(* CODESYS project CommonTypesAndFunctions.library
   Author: Stefan Dreyer
   Title: Common Helper for development
   Version: 1.0.0.0
   Placeholder: CommonTypsFunctions
   DocFormat: reStructuredText
   Description: Some things to collect...
      some based on OSCAT library.
      see www.oscat.de for here home
   Company: Stefan Dreyer
   LanguageModelAttribute: qualified-access-only
   DefaultNamespace: CommonTypesAndFunctions

Project tree, tasks and I/O mapping:
  libraries: CAA Types Extern, * (CAA Technical Workgroup); CAA Behaviour Model, * (CAA Technical Workgroup); CAA FB Factory, * (CAA Technical Workgroup); OSCAT NETWORK, 1.30 (OSCAT); SysSem, 3.5.5.0 (System); SysTypes Interfaces, 3.5.2.0 (System); BASIC, 3.3.3.0 (OSCAT); Time and Date, 3.5.7.0 (3S - Smart Software Solutions GmbH); CmpTls, 3.5.10.0 (System); SysProcess, 3.5.7.0 (System); SysTarget, 3.5.5.0 (System); SysMem, 3.5.12.0 (System); CmpX509Cert, 3.5.11.0 (System); CmpCrypto, 3.5.11.0 (System); MQTT, 1.1.0.0 (Stefan Dreyer); SysSocket2, 3.5.14.0 (System); SysSocket, 3.5.14.0 (System); Standard, 3.5.14.0 (System); CmpErrors2 Interfaces, 3.5.12.0 (System); Standard64, 3.5.13.0 (System)
  Common/
    Enums/
      data type ERROR
      data type VAR_TYPES
    Function Blocks/
      function block IP_CONTROL [ST]
      function block IP_CONTROL_135 [ST]
      function block IP_CONTROL_135_1 [ST]
      function block IP_CONTROL_old [ST]
      function block TIME_DATE_IMPULS [ST]
      function block TestString [ST]
      function block IP_CONTROL_TLS [ST]
      function block CounterToActuall [ST]: CounterInit, SetCounterResetImp
      function block StringImpact [ST]
      function block GetInstanceName [ST]: GetInstanceTopic
      function block RELAIS_OUT_16_TRANSLATOR [ST]
    Functions/
      function GET_DNS_IP [ST]
      function GetChar [ST]
      function find [ST]
      function len [ST]
      function concat [ST]
      function ResolveIPAddr [ST]
      function CheckDeltaValue [ST]
      function GetValueFromPointer [ST]
      function GetValueString [ST]
      function test [ST]
      function StrEquals [ST]
      function StrEqualsAtStart [ST]
      function GetValueFromStringPt [ST]
      function StrEqualsAtStartWithDelimiter [ST]
      function FindLastDot [ST]
      function MakeAllTypesPointer [ST]
      function GetJSONValue [ST]
    GlobalConstants/
      global variables MyConstants
    GlobalVariables/
      global variables Variables
    Interfaces/
    Structs/
    Templates/
      Behaviour Model/
        function block ETrigA_Temp [ST]: prvAbort, prvCyclicAction, prvResetOutputs, prvStart
        function block ETrigTlA_Temp [ST]: prvAbort, prvCyclicAction, prvResetOutputs, prvStart
        function block ETrigTl_Temp [ST]: prvAbort, prvCyclicAction, prvResetOutputs, prvStart
        function block ETrigToA_Temp [ST]: prvAbort, prvCyclicAction, prvResetOutputs, prvStart
        function block ETrigToTlA_Temp [ST]: prvAbort, prvCyclicAction, prvResetOutputs, prvStart
        function block ETrigToTl_Temp [ST]: prvAbort, prvCyclicAction, prvResetOutputs, prvStart
        function block ETrigTo_Temp [ST]: prvAbort, prvCyclicAction, prvResetOutputs, prvStart
        function block ETrig_Temp [ST]: prvAbort, prvCyclicAction, prvResetOutputs, prvStart
        function block LTrig_Temp [ST]: prvAbort, prvCyclicAction, prvResetOutputs, prvStart
      FB Factory/
        function block CustomData [ST]
        function block CustomFB [ST]: prvInstInit
        function block CustomFBFactory_heap [ST]: Create, prvInstCount, prvInstPoolExtendsFactor, prvInstSize
        function block CustomFBFactory_static [ST]: Create, prvInstPoolAdr, prvInstPoolSize, prvInstSize
    Types/
      data type ALL_TYPES_UNION
      data type ALL_TYPES_UNION_POINTER
      data type EEPROM_DATA
      data type IP_C
      data type TIME_DATE_IMPULS_DATA
      data type TLS_CONFIG
      data type PWConfigs
*)

// Common/Enums/ERROR
{attribute 'qualified_only'}
//{attribute 'conditionalshow'}
//{attribute 'conditionalshow' := 'SomeText'}
//{attribute 'hide'}
TYPE ERROR : (NO_ERROR, TIME_OUT); END_TYPE

// Common/Types/ALL_TYPES_UNION
TYPE ALL_TYPES_UNION :
UNION
	SINT_T:SINT;
	USINT_T:USINT;
	INT_T:INT;
	UINT_T:UINT;
	LINT_T:LINT;
	ULINT_T:ULINT;
	DINT_T:DINT;
	UDINT_T:UDINT;
	REAL_T:REAL;
	LREAL_T:LREAL;
	BYTE_T:BYTE;
	WORD_T:WORD;
	DWORD_T:DWORD;
	LWORD_T:LWORD;
	DT_T:DT;
	TIME_T:TIME;
	LTIME_T:LTIME;
	TOD_T:TOD;
	TOD_T2:ARRAY[0..1]OF TOD;
	DATE_T:DATE;
	BYTE_ARRAY:ARRAY[0..7]OF BYTE;
	BOOL_T:BOOL;
	//don't use strings UNION would be TO big....
END_UNION
END_TYPE

// Common/Types/ALL_TYPES_UNION_POINTER
TYPE ALL_TYPES_UNION_POINTER :
UNION
	POINTER_TO_SINT_T:POINTER TO SINT;
	POINTER_TO_USINT_T:POINTER TO USINT;
	POINTER_TO_INT_T:POINTER TO INT;
	POINTER_TO_UINT_T:POINTER TO UINT;
	POINTER_TO_LINT_T:POINTER TO LINT;
	POINTER_TO_ULINT_T:POINTER TO ULINT;
	POINTER_TO_DINT_T:POINTER TO DINT;
	POINTER_TO_UDINT_T:POINTER TO UDINT;
	POINTER_TO_REAL_T:POINTER TO REAL;
	POINTER_TO_LREAL_T:POINTER TO LREAL;
	POINTER_TO_BYTE_T:POINTER TO BYTE;
	POINTER_TO_WORD_T:POINTER TO WORD;
	POINTER_TO_DWORD_T:POINTER TO DWORD;
	POINTER_TO_LWORD_T:POINTER TO LWORD;
	POINTER_TO_DT_T:POINTER TO DT;
	POINTER_TO_TIME_T:POINTER TO TIME;
	POINTER_TO_LTIME_T:POINTER TO LTIME;
	POINTER_TO_TOD_T:POINTER TO TOD;
	POINTER_TO_TOD_T2:POINTER TO ARRAY[0..1]OF TOD;
	POINTER_TO_DATE_T:POINTER TO DATE;
	POINTER_TO_BYTE_ARRAY_T:POINTER TO ARRAY[0..7]OF BYTE;
	POINTER_TO_BOOL_T:POINTER TO BOOL;
	POINTER_TO_STRING_T: POINTER TO STRING(2000);
END_UNION
END_TYPE

// Common/Types/EEPROM_DATA
TYPE EEPROM_DATA :
STRUCT
	//FB_NO_AUTO:UINT;//auto createt FB NO, not possible because of multitasking ... so bad...
	FB_NO_IN:UINT;//allways check FB_IN_NO to be 0!!! so the EEPROM is free to do something!
	FB_NO_OUT:UINT;
	PAGE_IN:ARRAY[0..128-1] OF BYTE;
	PAGE_OUT:ARRAY[0..128-1] OF BYTE;
	READ_PAGE: BOOL;
	WRITE_PAGE: BOOL;
	ADDRESS_PAGE: UINT;
	ADDRESS_VALUE: UINT;
	VALUE_IN:ALL_TYPES_UNION;
	VALUE_OUT:ALL_TYPES_UNION; 
	READ_VALUE: BOOL;
	WRITE_VALUE: BOOL;
	PAGE_SIZE:UINT:=128;
	SIZE_OF_VALUE:UINT;
	SEMAPHORE:SysSem.RTS_IEC_HANDLE; //Semaphore for Consistence for EEPROM DATA is bus is out of main task
	HANDLE_VALID: BOOL;

END_STRUCT
END_TYPE

// Common/Types/IP_C
TYPE IP_C :
STRUCT
	C_MODE : BYTE;						(*W Mode: TCP/UCP AKTIV/PASSIV                               *)
	C_PORT : WORD;						(*W Portnummer                                               *)
	C_IP : DWORD;						(*W IP-Adresse gepackt wwxxyyzz = www.xxx.yyy.zzz            *)
	C_STATE : BYTE;						(*R Verbindungsstatus ON/OFF + Flanke ON/OFF                 *)
	C_ENABLE : BOOL;					(*W Freigabe für Connect                                     *)
	R_OBSERVE : BOOL;					(*W Empfang ueberwachen                                      *)
	TIME_RESET : BOOL;					(*W Alle Timer ruecksetzen                                   *)
	TLS: BOOL;							(*W Verbindung mit TLS		                                 *)
	

	ERROR : DWORD;					(*R vvwwxxyy (vv = CON_ERROR, ww = SEN_ERROR, xx = REC_ERROR *)
	FIFO : IP_FIFO_DATA;					(*I IP FIFO Struktur                                         *)
	MAILBOX : ARRAY [1..16] OF BYTE;	(*I Mailbox: Datenbereich für Bausteindatenaustausch         *)
END_STRUCT
END_TYPE

(* revision history
ks	18. oct. 2008	rev 1.1
	original version
*)

// Common/Types/TIME_DATE_IMPULS_DATA
TYPE TIME_DATE_IMPULS_DATA :
STRUCT
	
	IMP:BOOL;//1s impulse
	SYSTEM_TIME:DT;//Time on SYSTEM
	TIME_IO:BOOL;//TIME IS I.O.
	TD_TIME:OSCAT_BASIC.SDT;
	//impulse at 00:00:00
	DAY_CHANGE:BOOL;
END_STRUCT
END_TYPE

// Common/Types/TLS_CONFIG
TYPE TLS_CONFIG :
STRUCT
	//see CmpTls for Doku of Method, initialisied to work as client
	tlsMethod: CmpTls.CmpTlsMethod := CmpTlsMethod.TLSv2_CLIENT;
	//List of allowed ciphers, initialised to medium, see openSSL for cipherList config
	chiperList:STRING(255) := 'HIGH';
	//certificates and ca still not supportet by CmpTls. So initialised to dont use certificats....
	{info 'here to implement certificate use'}
	verifyMode:DWORD := CmpTlsConstants.TLS_VERIFY_CLIENT_ONCE;
	
END_STRUCT
END_TYPE

// Common/Enums/VAR_TYPES
{attribute 'qualified_only'}
{attribute 'strict'}
TYPE VAR_TYPES :
(
	//enum_member := 0
	SINT_T, USINT_T, INT_T, UINT_T, DINT_T, UDINT_T, 
				LINT_T, ULINT_T, REAL_T, LREAL_T, BYTE_T, WORD_T,
				DWORD_T, LWORD_T, DT_T, TIME_T, TOD_T, TOD2_T, DATE_T, ARRAY_T, BOOL_T,
				STRING_T, LTIME_T
);
END_TYPE

// Common/Types/PWConfigs
TYPE PWConfigs :
STRUCT
PointerTo:ALL_TYPES_UNION_POINTER;
//PointerTo1:POINTER TO BYTE;
ValueType:VAR_TYPES;
NeedsMQTT:BOOL;
NeedsDB:BOOL;
MQTTTopic:POINTER TO STRING;
MQTTName:POINTER TO STRING;
MQTTDiff:UINT;
MQTTDezimal:INT;
MQTTTime:TIME;
MQTTRetain:BOOL;
MQTTQoS:SD_MQTT.QoS;
DBName:STRING;
DBNum:UINT;




END_STRUCT
END_TYPE

// Common/GlobalConstants/MyConstants
{attribute 'qualified_only'}
//{attribute 'conditionalshow'}
//{attribute 'conditionalshow' := 'SomeText'}
//{attribute 'hide'}
VAR_GLOBAL CONSTANT
	gc_iDummy : INT := 42; /// This is a dummy global constant variable
	//Countrs in coutr ;)
	COUNTER_COUNT:UINT:=5;
END_VAR

// Common/GlobalVariables/Variables
{attribute 'qualified_only'}
//{attribute 'conditionalshow'}
//{attribute 'conditionalshow' := 'SomeText'}
//{attribute 'hide'}
VAR_GLOBAL
	g_iDummy : INT; /// This is a dummy global variable
END_VAR

// Common/Templates/Behaviour Model/ETrigA_Temp
//{attribute 'hide_all_locals'}
//{attribute 'conditionalshow_all_locals' := 'SomeText'}
//{attribute 'conditionalshow_all_locals'}
//{attribute 'conditionalshow' := 'SomeText'}
//{attribute 'conditionalshow'}
//{attribute 'hide'}
FUNCTION_BLOCK ETrigA_Temp EXTENDS CBM.ETrigA
VAR_INPUT
	(* specific Inputs *)
END_VAR
VAR_OUTPUT
	eError : ERROR;
	(* specific Outputs *)
END_VAR
VAR
	(* specific vars *)
END_VAR

SUPER^();
IF iError = CBM.ERROR.TIME_OUT THEN
	eError := ERROR.TIME_OUT;
ELSE
	eError := iError;
END_IF

{attribute 'hide'}
METHOD prvAbort : BOOL
VAR_INPUT
END_VAR
VAR
END_VAR
IF xError THEN (* abort because of error *)
	(* TODO: insert specific Code here *)
ELSE (* user abort *)
	(* TODO: insert specific Code here *)
END_IF
xAbortInProgress:= FALSE;
END_METHOD

{attribute 'hide'}
METHOD prvCyclicAction : BOOL
VAR_INPUT
END_VAR
VAR
END_VAR
(* TODO: insert specific Code here *)
xDone:= TRUE;
(* if an error occurs, set iError to a value else than zero instead of xDone:= TRUE *)
(* to keep repeat loop *)
END_METHOD

{attribute 'hide'}
METHOD prvResetOutputs : BOOL
VAR_INPUT
END_VAR
VAR
END_VAR
(* TODO: insert specific Code here *)
SUPER^.prvResetOutputs();
END_METHOD

{attribute 'hide'}
METHOD prvStart : BOOL
VAR_INPUT
END_VAR
VAR
END_VAR
(* this code is called, when the application is started (rising edge of xExecute *)
(* TODO: copy specific input variables into local copies *)
(* TODO: insert specific Code here *)
;
END_METHOD

END_FUNCTION_BLOCK

// Common/Templates/Behaviour Model/ETrigTlA_Temp
//{attribute 'hide_all_locals'}
//{attribute 'conditionalshow_all_locals' := 'SomeText'}
//{attribute 'conditionalshow_all_locals'}
//{attribute 'conditionalshow' := 'SomeText'}
//{attribute 'conditionalshow'}
//{attribute 'hide'}
FUNCTION_BLOCK ETrigTlA_Temp EXTENDS CBM.ETrigTlA
VAR_INPUT
	(* specific Inputs *)
END_VAR
VAR_OUTPUT
	eError : ERROR;
	(* specific Outputs *)
END_VAR
VAR
	(* specific vars *)
END_VAR

SUPER^();
IF iError = CBM.ERROR.TIME_OUT THEN
	eError := ERROR.TIME_OUT;
ELSE
	eError := iError;
END_IF

{attribute 'hide'}
METHOD prvAbort : BOOL
VAR_INPUT
END_VAR
VAR
END_VAR
IF xError THEN (* abort because of error *)
	(* TODO: insert specific Code here *)
ELSE (* user abort *)
	(* TODO: insert specific Code here *)
END_IF
xAbortInProgress:= FALSE;
END_METHOD

{attribute 'hide'}
METHOD prvCyclicAction : BOOL
VAR_INPUT
END_VAR
VAR
END_VAR
(* TODO: insert specific Code here *)
xDone:= TRUE;
(* if an error occurs, set iError to a value else than zero instead of xDone:= TRUE *)
(* to keep repeat loop *)
END_METHOD

{attribute 'hide'}
METHOD prvResetOutputs : BOOL
VAR_INPUT
END_VAR
VAR
END_VAR
(* TODO: insert specific Code here *)
SUPER^.prvResetOutputs();
END_METHOD

{attribute 'hide'}
METHOD prvStart : BOOL
VAR_INPUT
END_VAR
VAR
END_VAR
(* this code is called, when the application is started (rising edge of xExecute *)
(* TODO: copy specific input variables into local copies *)
(* TODO: insert specific Code here *)
;
END_METHOD

END_FUNCTION_BLOCK

// Common/Templates/Behaviour Model/ETrigTl_Temp
//{attribute 'hide_all_locals'}
//{attribute 'conditionalshow_all_locals' := 'SomeText'}
//{attribute 'conditionalshow_all_locals'}
//{attribute 'conditionalshow' := 'SomeText'}
//{attribute 'conditionalshow'}
//{attribute 'hide'}
FUNCTION_BLOCK ETrigA_Temp EXTENDS CBM.ETrigTl
VAR_INPUT
	(* specific Inputs *)
END_VAR
VAR_OUTPUT
	eError : ERROR;
	(* specific Outputs *)
END_VAR
VAR
	(* specific vars *)
END_VAR

SUPER^();
IF iError = CBM.ERROR.TIME_OUT THEN
	eError := ERROR.TIME_OUT;
ELSE
	eError := iError;
END_IF

{attribute 'hide'}
METHOD prvAbort : BOOL
VAR_INPUT
END_VAR
VAR
END_VAR
IF xError THEN (* abort because of error *)
	(* TODO: insert specific Code here *)
ELSE (* user abort *)
	(* TODO: insert specific Code here *)
END_IF
xAbortInProgress:= FALSE;
END_METHOD

{attribute 'hide'}
METHOD prvCyclicAction : BOOL
VAR_INPUT
END_VAR
VAR
END_VAR
(* TODO: insert specific Code here *)
xDone:= TRUE;
(* if an error occurs, set iError to a value else than zero instead of xDone:= TRUE *)
(* to keep repeat loop *)
END_METHOD

{attribute 'hide'}
METHOD prvResetOutputs : BOOL
VAR_INPUT
END_VAR
VAR
END_VAR
(* TODO: insert specific Code here *)
SUPER^.prvResetOutputs();
END_METHOD

{attribute 'hide'}
METHOD prvStart : BOOL
VAR_INPUT
END_VAR
VAR
END_VAR
(* this code is called, when the application is started (rising edge of xExecute *)
(* TODO: copy specific input variables into local copies *)
(* TODO: insert specific Code here *)
;
END_METHOD

END_FUNCTION_BLOCK

// Common/Templates/Behaviour Model/ETrigToA_Temp
//{attribute 'hide_all_locals'}
//{attribute 'conditionalshow_all_locals' := 'SomeText'}
//{attribute 'conditionalshow_all_locals'}
//{attribute 'conditionalshow' := 'SomeText'}
//{attribute 'conditionalshow'}
//{attribute 'hide'}
FUNCTION_BLOCK ETrigToA_Temp EXTENDS CBM.ETrigToA
VAR_INPUT
	(* specific Inputs *)
END_VAR
VAR_OUTPUT
	eError : ERROR;
	(* specific Outputs *)
END_VAR
VAR
	(* specific vars *)
END_VAR

SUPER^();
IF iError = CBM.ERROR.TIME_OUT THEN
	eError := ERROR.TIME_OUT;
ELSE
	eError := iError;
END_IF

{attribute 'hide'}
METHOD prvAbort : BOOL
VAR_INPUT
END_VAR
VAR
END_VAR
IF xError THEN (* abort because of error *)
	(* TODO: insert specific Code here *)
ELSE (* user abort *)
	(* TODO: insert specific Code here *)
END_IF
xAbortInProgress:= FALSE;
END_METHOD

{attribute 'hide'}
METHOD prvCyclicAction : BOOL
VAR_INPUT
END_VAR
VAR
END_VAR
(* TODO: insert specific Code here *)
xDone:= TRUE;
(* if an error occurs, set iError to a value else than zero instead of xDone:= TRUE *)
END_METHOD

{attribute 'hide'}
METHOD prvResetOutputs : BOOL
VAR_INPUT
END_VAR
VAR
END_VAR
(* TODO: insert specific Code here *)
SUPER^.prvResetOutputs();
END_METHOD

{attribute 'hide'}
METHOD prvStart : BOOL
VAR_INPUT
END_VAR
VAR
END_VAR
(* this code is called, when the application is started (rising edge of xExecute *)
(* TODO: copy specific input variables into local copies *)
(* TODO: insert specific Code here *)
;
END_METHOD

END_FUNCTION_BLOCK

// Common/Templates/Behaviour Model/ETrigToTlA_Temp
//{attribute 'hide_all_locals'}
//{attribute 'conditionalshow_all_locals' := 'SomeText'}
//{attribute 'conditionalshow_all_locals'}
//{attribute 'conditionalshow' := 'SomeText'}
//{attribute 'conditionalshow'}
//{attribute 'hide'}
FUNCTION_BLOCK ETrigToTlA_Temp EXTENDS CBM.ETrigToTlA
VAR_INPUT
	(* specific Inputs *)
END_VAR
VAR_OUTPUT
	eError : ERROR;
	(* specific Outputs *)
END_VAR
VAR
	(* specific vars *)
END_VAR

SUPER^();
IF iError = CBM.ERROR.TIME_OUT THEN
	eError := ERROR.TIME_OUT;
ELSE
	eError := iError;
END_IF

{attribute 'hide'}
METHOD prvAbort : BOOL
VAR_INPUT
END_VAR
VAR
END_VAR
IF xError THEN (* abort because of error *)
	(* TODO: insert specific Code here *)
ELSE (* user abort *)
	(* TODO: insert specific Code here *)
END_IF
xAbortInProgress:= FALSE;
END_METHOD

{attribute 'hide'}
METHOD prvCyclicAction : BOOL
VAR_INPUT
END_VAR
VAR
END_VAR
(* TODO: insert specific Code here *)
xDone:= TRUE;
(* if an error occurs, set iError to a value else than zero instead of xDone:= TRUE *)
(* to keep repeat loop *)
END_METHOD

{attribute 'hide'}
METHOD prvResetOutputs : BOOL
VAR_INPUT
END_VAR
VAR
END_VAR
(* TODO: insert specific Code here *)
SUPER^.prvResetOutputs();
END_METHOD

{attribute 'hide'}
METHOD prvStart : BOOL
VAR_INPUT
END_VAR
VAR
END_VAR
(* this code is called, when the application is started (rising edge of xExecute *)
(* TODO: copy specific input variables into local copies *)
(* TODO: insert specific Code here *)
;
END_METHOD

END_FUNCTION_BLOCK

// Common/Templates/Behaviour Model/ETrigToTl_Temp
//{attribute 'hide_all_locals'}
//{attribute 'conditionalshow_all_locals' := 'SomeText'}
//{attribute 'conditionalshow_all_locals'}
//{attribute 'conditionalshow' := 'SomeText'}
//{attribute 'conditionalshow'}
//{attribute 'hide'}
FUNCTION_BLOCK ETrigToTl_Temp EXTENDS CBM.ETrigToTl
VAR_INPUT
	(* specific Inputs *)
END_VAR
VAR_OUTPUT
	eError : ERROR;
	(* specific Outputs *)
END_VAR
VAR
	(* specific vars *)
END_VAR

SUPER^();
IF iError = CBM.ERROR.TIME_OUT THEN
	eError := ERROR.TIME_OUT;
ELSE
	eError := iError;
END_IF

{attribute 'hide'}
METHOD prvAbort : BOOL
VAR_INPUT
END_VAR
VAR
END_VAR
IF xError THEN (* abort because of error *)
	(* TODO: insert specific Code here *)
ELSE (* user abort *)
	(* TODO: insert specific Code here *)
END_IF
xAbortInProgress:= FALSE;
END_METHOD

{attribute 'hide'}
METHOD prvCyclicAction : BOOL
VAR_INPUT
END_VAR
VAR
END_VAR
(* TODO: insert specific Code here *)
xDone:= TRUE;
(* if an error occurs, set iError to a value else than zero instead of xDone:= TRUE *)
(* to keep repeat loop *)
END_METHOD

{attribute 'hide'}
METHOD prvResetOutputs : BOOL
VAR_INPUT
END_VAR
VAR
END_VAR
(* TODO: insert specific Code here *)
SUPER^.prvResetOutputs();
END_METHOD

{attribute 'hide'}
METHOD prvStart : BOOL
VAR_INPUT
END_VAR
VAR
END_VAR
(* this code is called, when the application is started (rising edge of xExecute *)
(* TODO: copy specific input variables into local copies *)
(* TODO: insert specific Code here *)
;
END_METHOD

END_FUNCTION_BLOCK

// Common/Templates/Behaviour Model/ETrigTo_Temp
//{attribute 'hide_all_locals'}
//{attribute 'conditionalshow_all_locals' := 'SomeText'}
//{attribute 'conditionalshow_all_locals'}
//{attribute 'conditionalshow' := 'SomeText'}
//{attribute 'conditionalshow'}
//{attribute 'hide'}
FUNCTION_BLOCK ETrigTo_Temp EXTENDS CBM.ETrigTo
VAR_INPUT
	(* specific Inputs *)
END_VAR
VAR_OUTPUT
	eError : ERROR;
	(* specific Outputs *)
END_VAR
VAR
	(* specific vars *)
END_VAR

SUPER^();
IF iError = CBM.ERROR.TIME_OUT THEN
	eError := ERROR.TIME_OUT;
ELSE
	eError := iError;
END_IF

{attribute 'hide'}
METHOD prvAbort : BOOL
VAR_INPUT
END_VAR
VAR
END_VAR
IF xError THEN (* abort because of error *)
	(* TODO: insert specific Code here *)
ELSE (* user abort *)
	(* TODO: insert specific Code here *)
END_IF
xAbortInProgress:= FALSE;
END_METHOD

{attribute 'hide'}
METHOD prvCyclicAction : BOOL
VAR_INPUT
END_VAR
VAR
END_VAR
(* TODO: insert specific Code here *)
xDone:= TRUE;
(* if an error occurs, set iError to a value else than zero instead of xDone:= TRUE *)
(* to keep repeat loop *)
END_METHOD

{attribute 'hide'}
METHOD prvResetOutputs : BOOL
VAR_INPUT
END_VAR
VAR
END_VAR
(* TODO: insert specific Code here *)
SUPER^.prvResetOutputs();
END_METHOD

{attribute 'hide'}
METHOD prvStart : BOOL
VAR_INPUT
END_VAR
VAR
END_VAR
(* this code is called, when the application is started (rising edge of xExecute *)
(* TODO: copy specific input variables into local copies *)
(* TODO: insert specific Code here *)
;
END_METHOD

END_FUNCTION_BLOCK

// Common/Templates/Behaviour Model/ETrig_Temp
//{attribute 'hide_all_locals'}
//{attribute 'conditionalshow_all_locals' := 'SomeText'}
//{attribute 'conditionalshow_all_locals'}
//{attribute 'conditionalshow' := 'SomeText'}
//{attribute 'conditionalshow'}
//{attribute 'hide'}
FUNCTION_BLOCK ETrig_Temp EXTENDS CBM.ETrig
VAR_INPUT
	(* specific Inputs *)
END_VAR
VAR_OUTPUT
	eError : ERROR;
	(* specific Outputs *)
END_VAR
VAR
	(* specific vars *)
END_VAR

SUPER^();
IF iError = CBM.ERROR.TIME_OUT THEN
	eError := ERROR.TIME_OUT;
ELSE
	eError := iError;
END_IF

{attribute 'hide'}
METHOD prvAbort : BOOL
VAR_INPUT
END_VAR
VAR
END_VAR
IF xError THEN (* abort because of error *)
	(* TODO: insert specific Code here *)
ELSE (* user abort *)
	(* TODO: insert specific Code here *)
END_IF
xAbortInProgress:= FALSE;
END_METHOD

{attribute 'hide'}
METHOD prvCyclicAction : BOOL
VAR_INPUT
END_VAR
VAR
END_VAR
(* TODO: insert specific Code here *)
xDone:= TRUE;
(* if an error occurs, set iError to a value else than zero instead of xDone:= TRUE *)
(* to keep repeat loop *)
END_METHOD

{attribute 'hide'}
METHOD prvResetOutputs : BOOL
VAR_INPUT
END_VAR
VAR
END_VAR
(* TODO: insert specific Code here *)
SUPER^.prvResetOutputs();
END_METHOD

{attribute 'hide'}
METHOD prvStart : BOOL
VAR_INPUT
END_VAR
VAR
END_VAR
(* this code is called, when the application is started (rising edge of xExecute *)
(* TODO: copy specific input variables into local copies *)
(* TODO: insert specific Code here *)
;
END_METHOD

END_FUNCTION_BLOCK

// Common/Templates/Behaviour Model/LTrig_Temp
//{attribute 'hide_all_locals'}
//{attribute 'conditionalshow_all_locals' := 'SomeText'}
//{attribute 'conditionalshow_all_locals'}
//{attribute 'conditionalshow' := 'SomeText'}
//{attribute 'conditionalshow'}
//{attribute 'hide'}
FUNCTION_BLOCK LTrig_Temp EXTENDS CBM.LTrig
VAR_INPUT
	(* specific Inputs *)
END_VAR
VAR_OUTPUT
	eError : ERROR;
	(* specific Outputs *)
END_VAR
VAR
	(* specific vars *)
END_VAR

SUPER^();
IF iError = CBM.ERROR.TIME_OUT THEN
	eError := ERROR.TIME_OUT;
ELSE
	eError := iError;
END_IF

{attribute 'hide'}
METHOD prvAbort : BOOL
VAR_INPUT
END_VAR
VAR
END_VAR
IF xError THEN (* abort because of error *)
	(* TODO: insert specific Code here *)
ELSE (* user abort *)
	(* TODO: insert specific Code here *)
END_IF
xAbortInProgress:= FALSE;
END_METHOD

{attribute 'hide'}
METHOD prvCyclicAction : BOOL
VAR_INPUT
END_VAR
VAR
END_VAR
(* TODO: insert specific Code here *)
xDone:= TRUE;
(* if an error occurs, set iError to a value else than zero instead of xDone:= TRUE *)
(* to keep repeat loop *)
END_METHOD

{attribute 'hide'}
METHOD prvResetOutputs : BOOL
VAR_INPUT
END_VAR
VAR
END_VAR
(* TODO: insert specific Code here *)
SUPER^.prvResetOutputs();
END_METHOD

{attribute 'hide'}
METHOD prvStart : BOOL
VAR_INPUT
END_VAR
VAR
END_VAR
(* this code is called, when the application is started (rising edge of xExecute *)
(* TODO: copy specific input variables into local copies *)
(* TODO: insert specific Code here *)
;
END_METHOD

END_FUNCTION_BLOCK

// Common/Templates/FB Factory/CustomData
// This is a container to carry init data from the Create methode of the factory
// to the prvInstInit methode of the new generated function block instance
{attribute 'enable_dynamic_creation'}
//{attribute 'hide_all_locals'}
//{attribute 'conditionalshow_all_locals' := 'SomeText'}
//{attribute 'conditionalshow_all_locals'}
//{attribute 'conditionalshow' := 'SomeText'}
//{attribute 'conditionalshow'}
//{attribute 'hide'}
FUNCTION_BLOCK CustomData EXTENDS FBF.InstanceData
VAR_INPUT
	(* Todo: Add your application specific data as input variables *)
END_VAR

(* !! Do not add any executable code here !! *)
SUPER^();

END_FUNCTION_BLOCK

// Common/Templates/FB Factory/CustomFB
{attribute 'enable_dynamic_creation'}
//{attribute 'hide_all_locals'}
//{attribute 'conditionalshow_all_locals' := 'SomeText'}
//{attribute 'conditionalshow_all_locals'}
//{attribute 'conditionalshow' := 'SomeText'}
//{attribute 'conditionalshow'}
//{attribute 'hide'}
FUNCTION_BLOCK CustomFB EXTENDS FBF.InstanceBase;
VAR_INPUT
END_VAR
VAR_OUTPUT
END_VAR
VAR
END_VAR

SUPER^();

// This methode is called from the factory to give a chance
// to initialize the new fb instance with the content of itfData
//{attribute 'hide_all_locals'}
//{attribute 'conditionalshow_all_locals' := 'SomeText'}
//{attribute 'conditionalshow_all_locals'}
//{attribute 'conditionalshow' := 'SomeText'}
//{attribute 'conditionalshow'}
//{attribute 'hide'}
METHOD prvInstInit : FBF.ERROR
VAR_INPUT
	itfData : FBF.IData; 
END_VAR
VAR
	pData : POINTER TO CustomData;
	xOk : BOOL;
END_VAR
SUPER^.prvInstInit(itfData);
xOk := __QUERYPOINTER(itfData, pData);
IF xOk THEN
	(* THIS^.iLocalVar := pData^.iInitValue *);
END_IF
END_METHOD

END_FUNCTION_BLOCK

// Common/Templates/FB Factory/CustomFBFactory_heap
// This is a template for a factory with an heap based extendable memory pool
{attribute 'enable_dynamic_creation'}
//{attribute 'hide_all_locals'}
//{attribute 'conditionalshow_all_locals' := 'SomeText'}
//{attribute 'conditionalshow_all_locals'}
//{attribute 'conditionalshow' := 'SomeText'}
//{attribute 'conditionalshow'}
//{attribute 'hide'}
FUNCTION_BLOCK CustomFBFactory_heap EXTENDS FBF.FactoryBase
VAR
END_VAR

SUPER^();

(* Please replace CustonFB with your specific function block type *)
(* There is no need to change anything else !!! *)
METHOD Create : POINTER TO CustomFB
VAR_INPUT
	itfData : FBF.IData;
END_VAR
VAR_OUTPUT
	eError : FBF.ERROR;
END_VAR
VAR
	hInst : CAA.HANDLE;
	itfInst : FBF.IInstance;
	xOk : BOOL;
END_VAR
(* !!! This code must not be subject to change !!! *)
hInst := SUPER^.prvAllocInstMem(eError => eError);
Create := SUPER^.prvGetInstPointer(hInst);
IF Create <> 0 AND eError = FBF.ERROR.NO_ERROR THEN

	{implicit on}
	Create^.__vfInit();
	Create^.FB_Init(TRUE, FALSE);
	{implicit off}

	xOk := __QUERYINTERFACE(Create^, itfInst);
	IF xOk THEN
		xOk := SUPER^.prvInstInit(itfInst, hInst, itfData, eError=>eError);
	ELSE
		eError := FBF.ERROR.WRONG_INTERFACE;
	END_IF

	IF NOT xOk THEN
		SUPER^.prvFreeInstMem(hInst);
		Create := CAA.gc_pNULL;
	END_IF
END_IF
END_METHOD

//{attribute 'conditionalshow' := 'SomeText'}
//{attribute 'conditionalshow'}
//{attribute 'hide'}
PROPERTY prvInstCount : CAA.COUNT (* ctInst *)
GET
(* Please choose a proper value for prvInstCount *)
prvInstCount := 10;
END_GET
END_PROPERTY

//{attribute 'conditionalshow' := 'SomeText'}
//{attribute 'conditionalshow'}
//{attribute 'hide'}
PROPERTY prvInstPoolExtendsFactor : USINT (* usiFactor [0..x%] *)
GET
(* Please choose a proper value for prvInstPoolExtendsFactor *)
(* This value will be interpreted as a 0..x% size extendsion related to the original size of the pool *)
prvInstPoolExtendsFactor := 20;
END_GET
END_PROPERTY

//{attribute 'conditionalshow' := 'SomeText'}
//{attribute 'conditionalshow'}
//{attribute 'hide'}
PROPERTY prvInstSize : CAA.SIZE (* szInst *)
GET
(* Please replace CustomFB with your specific function block type *)
prvInstSize := sizeof(CustomFB);
END_GET
END_PROPERTY

END_FUNCTION_BLOCK

// Common/Templates/FB Factory/CustomFBFactory_static
// This is a template for a factory with an static iec memory based memory pool which a fixed capacity
{attribute 'enable_dynamic_creation'}
//{attribute 'hide_all_locals'}
//{attribute 'conditionalshow_all_locals' := 'SomeText'}
//{attribute 'conditionalshow_all_locals'}
//{attribute 'conditionalshow' := 'SomeText'}
//{attribute 'conditionalshow'}
//{attribute 'hide'}
FUNCTION_BLOCK CustomFBFactory_static EXTENDS FBF.FactoryBase
VAR
	// Please change the size of abyPoolMemory with your specific application need
	abyPoolMemory : ARRAY[0..529] OF BYTE;
END_VAR

SUPER^();

(* Please replace CustonFB with our specific function block type *)
(* There is no need to change anything else !!! *)
METHOD Create : POINTER TO CustomFB
VAR_INPUT
	itfData : FBF.IData;
END_VAR
VAR_OUTPUT
	eError : FBF.ERROR;
END_VAR
VAR
	hInst : CAA.HANDLE;
	itfInst : FBF.IInstance;
	xOk : BOOL;
END_VAR
(* !!! This code must not be subject to change !!! *)
hInst := SUPER^.prvAllocInstMem(eError => eError);
Create := SUPER^.prvGetInstPointer(hInst);
IF Create <> 0 AND eError = FBF.ERROR.NO_ERROR THEN

	{implicit on}
	Create^.__vfInit();
	Create^.FB_Init(TRUE, FALSE);
	{implicit off}

	xOk := __QUERYINTERFACE(Create^, itfInst);
	IF xOk THEN
		xOk := SUPER^.prvInstInit(itfInst, hInst, itfData, eError=>eError);
	ELSE
		eError := FBF.ERROR.WRONG_INTERFACE;
	END_IF

	IF NOT xOk THEN
		SUPER^.prvFreeInstMem(hInst);
		Create := CAA.gc_pNULL;
	END_IF
END_IF
END_METHOD

//{attribute 'conditionalshow' := 'SomeText'}
//{attribute 'conditionalshow'}
//{attribute 'hide'}
PROPERTY prvInstPoolAdr : CAA.PVOID (* pPool *)
GET
prvInstPoolAdr := ADR(abyPoolMemory);
END_GET
END_PROPERTY

//{attribute 'conditionalshow' := 'SomeText'}
//{attribute 'conditionalshow'}
//{attribute 'hide'}
PROPERTY prvInstPoolSize : CAA.SIZE (* szPool *)
GET
prvInstPoolSize := sizeof(abyPoolMemory);
END_GET
END_PROPERTY

//{attribute 'conditionalshow' := 'SomeText'}
//{attribute 'conditionalshow'}
//{attribute 'hide'}
PROPERTY prvInstSize : CAA.SIZE (* szInst *)
GET
(* Please replace CustomFB with your specific function block type *)
prvInstSize := sizeof(CustomFB);
END_GET
END_PROPERTY

END_FUNCTION_BLOCK

// Common/Function Blocks/IP_CONTROL
FUNCTION_BLOCK IP_CONTROL
VAR_IN_OUT
	IP_C : IP_C; (* IP_Control Verwaltungsstruktur *)
	S_BUF : NETWORK_BUFFER; (* Externer Sendbuffer *)
	R_BUF : NETWORK_BUFFER; (* Externer Receivebuffer *)
END_VAR
VAR_INPUT
	IP : DWORD; (* IP Adresse *)
	PORT : WORD; (* Port Nummer *)
	TIME_OUT : TIME; (* Ueberwachungszeit Connect / Send / Receive *)

END_VAR
VAR
	TLS_CONFIG:POINTER TO TLS_CONFIG;
	c_time : UDINT; (* CONNECT-Time (Zeit bei nicht vorhandener Verbindung) *)
	s_time : UDINT; (* SEND-Time    (Zeit seit letzten Datensenden) *)
	r_time : UDINT; (* RECEIVE-Time (Zeit seit letztem Datenempfang) *)

	c_enable : BOOL; (* Connect: freigabe *)
	c_ip : DWORD; (* Connect: aktuelle IP-Adresse *)
	c_port : WORD; (* Connect: aktuelle Port-Nummer *)
	c_mode : BYTE; (* Connect: aktueller Mode UDP/TCP...... *)
	c_status : BYTE; (* Connect: Status (Errorcode) *)
	c_ready : BOOL; (* Connect: Verbindung aufgebaut *)
	c_ready_old : BOOL; (* Connect: letzter Zustand von c_ready für Flankenauswertung *)
	c_select : BOOL; (* non blocking mode - abfrage über select durchführen *)
	c_fdWrite :  SOCKET_FD_SET;
	c_Timeout : SOCKET_TIMEVAL;
	//use a TLS connection
	TLS: BOOL;

		
	s_total : INT; (* Send: Gesamtanzahl Bytes zum senden *)
	s_cur_pos : INT; (* Send: aktuelle Sendeposition *)
	s_cur_size : INT; (* Send: aktuelle Sendegroesse *)
	s_max_size : INT; (* Send: maximale Telegrammlänge fuer Senden *)
	s_start : BOOL; (* Send: Sende modus aktivieren *)
	s_active : BOOL; (* Send: Daten senden ist aktiv *)
	s_req : BOOL; (* Send: Start Daten senden *)
	s_done : BOOL; (* Send: ohne Fehler beendet *)
	s_status : BYTE; (* Send: Status (Errorcodes) *)

	r_status : BYTE; (* Receive: Status (Errorcodes) *)
	r_count : INT; (* Receive: Anzahl empfangener Bytes *)
	r_offset : INT; (* Receive: aktuelle Position in externen Receivebuffer *)
	r_max_size : INT; (* Receive: groesse des externen Empfangbuffers*)

	new_connection : BOOL; (* Neue Verbindungsparameter vorhanden *)
	tx : DWORD; (* letzter zeitwert *)
	error_time : DWORD; (* aktueller Timeout-Wert *)
	//Socket Parameter
	SysSockParameter:SysSocket2.SysSocket2_Parameter;
	SysSockSpec : SysSocket2.SysSocket2_SpecificParameter;
	state: BYTE; (* schrittmerker für connect *)
	server_socket : RTS_IEC_HANDLE:= RTS_INVALID_HANDLE;                // Handle Pointing to our Socket
	socket : RTS_IEC_HANDLE:= RTS_INVALID_HANDLE;
	//TlsHandle := RTS_IEC_HANDLE:= RTS_INVALID_HANDLE;
	//server_socket : DINT:= RTS_INVALID_HANDLE;
	//socket : DINT:= RTS_INVALID_HANDLE;
	sockaddr : SOCKADDRESS;
	sockaddr_size : DWORD;
	plc_841 : BOOL;
	plc_881 : BOOL;
	dint_true : DINT := 1;
	dint_false : DINT := 0;
	bytes_received : DINT;
	bytes_sent : DINT;
	udp_mode : BOOL;

	pResult : RTS_IEC_RESULT; //Needed for V3 Lib
	FunctionResult 	: UDINT ;   
  	tAddress                	: INADDR;                           // Strucutre to define our internet address
	TESTtAddress               	: INADDR;   
	(*LOG_MSG : LOG_MSG;
	_debug_enable : BOOL := TRUE;
	debug_index : INT;
	debug_ID : INT;
	debug_lasterror : DWORD;
	debug_last_id : INT := 255;
	state_last: BYTE;*)
	
	TlsConnectTime:DWORD;
	TlsConnectLastTick:DWORD;
		
END_VAR

VAR CONSTANT
	STOP : BYTE := 0;
	TS_INIT: BYTE := 1;
	TS_OPEN : BYTE:= 2;

	UDP_INIT : BYTE:= 31;

	TC_INIT : BYTE:= 51;
	TC_CONNECT : BYTE:= 52;

	C_WAIT : BYTE:= 250;
	C_CLOSE : BYTE:= 251;
	

END_VAR

(*

version 1.9		26. Feb. 2012
programmer 		ks
tested by			ks

IP_CONTROL ist ein Wrapper-Baustein um eine Hersteller neutrale Schnittstelle zum Ethernet zu schaffen
*)

(* ---------------------- Debug-Message ----------------------------*)
(*IF _debug_enable THEN
	IF IP_C.FIFO.ID > BYTE#0 THEN (* nur wenn Teilnehmer ID's vorhanden sind *)
		debug_index := IP_C.FIFO.NR;
		debug_ID := BYTE_TO_INT(IP_C.FIFO.X[debug_index]);
	END_IF;
END_IF;*)
(* -----------------------------------------------------------------------------*)

(* read system time *)
tx := OSCAT_BASIC.T_PLC_MS();

IF IP_C.C_PORT = 0 THEN
	IP_C.C_PORT := PORT; (* uebergebenen PORT durch parametrierten PORT ersetzen *)
END_IF;
IF IP_C.C_IP = 0 AND IP_C.C_MODE < 4 THEN
	IP_C.C_IP := IP; (* uebergebene IP durch paramtrierte IP ersetzen *)
END_IF;

new_connection := c_ip <> IP_C.C_IP OR c_mode <> (IP_C.C_MODE AND 2#1111111) OR c_port <> IP_C.C_PORT; (* neue Verbindungs erwünscht ? *)
c_enable := IP_C.C_ENABLE AND NOT new_connection;

IF IP_C.C_ENABLE AND IP_C.ERROR = 0 AND state = STOP THEN (* Freigabe,kein Fehler,kein Socket offen *)
	c_ip   := IP_C.C_IP;
	c_mode := IP_C.C_MODE AND 2#1111111; //bit 7 for TLS Mode
	//TLS := IP_C.C_MODE.7;
	c_port := IP_C.C_PORT;
	plc_841 := ADR(%MW0)=16#30000000; (*750-841*)
	plc_881 := ADR(%MW0)=16#20000000; (*750-881*)
	udp_mode := C_MODE.0; (* Mode 1,3,5 = udp *)

	error_time := TIME_TO_DWORD(MAX(T#200ms,TIME_OUT));
	IP_C.TIME_RESET := TRUE; (* Alle Timer ruecksetzen *)

	r_max_size := UINT_TO_INT(SIZEOF(R_BUF.BUFFER));
	s_max_size := UINT_TO_INT(SIZEOF(S_BUF.BUFFER));

	IF C_MODE.0 THEN (* Mode: 1,3,5 = UDP CLIENT/SERVER *)
		state := UDP_INIT;
	ELSIF C_MODE = 0 THEN (* Mode: 0 = TCP CLIENT *)
		state := TC_INIT;
	ELSE
		state := TS_INIT; (* Mode: 2,4 = TCP SERVER *)
	END_IF;

	(* ---------------------- Debug-Message ----------------------------*)
	(*IF _debug_enable THEN
		LOG_CL.NEW_MSG := 'IP_CON: MODE ~1 / IP ~2 / PORT ~3 /ID ~6';
		LOG_CL.PRINTF[1] := BYTE_TO_STRING(C_MODE);
		LOG_CL.PRINTF[2] := IP4_TO_STRING(c_ip);
		LOG_CL.PRINTF[3] := WORD_TO_STRING(c_port);
		LOG_CL.PRINTF[6] := INT_TO_STRING(debug_ID);
		LOG_MSG();
	END_IF;*)
	(* -----------------------------------------------------------------------------*)

END_IF;

(* ---------------------- Debug-Message ----------------------------*)
(*IF  _debug_enable THEN
	IF state <> state_last THEN
		LOG_CL.NEW_MSG := 'IP_STEP ~1 -IP_ID ~6';
		LOG_CL.PRINTF[1] := BYTE_TO_STRING(state);
		LOG_CL.PRINTF[6] := INT_TO_STRING(debug_ID);
		LOG_MSG();
		state_last := state;
	END_IF;
END_IF;*)
(* -----------------------------------------------------------------------------*)

IF IP_C.TIME_RESET THEN (* Alle Timer ruecksetzen *)
	IP_C.TIME_RESET := FALSE; (* Reset rücksetzen *)
	c_time := tx; (* Connect Timer ruecksetzen *)
	s_time := tx; (* Send Timer ruecksetzen *)
	r_time := tx; (* Receive Timer ruecksetzen *)

	c_status := BYTE#0; (* letzten Connect Fehler rücksetzen *)
	s_status := BYTE#0; (* letzten Send Fehler rücksetzen *)
	r_status := BYTE#0; (* letzten Receive Fehler rücksetzen *)
END_IF;

(* ---------------------------------------------- *)

CASE state OF

UDP_INIT: (* UDP_CLIENT + SERVER *)
	//socket := SysSock2Create(SOCKET_AF_INET, SOCKET_DGRAM, SOCKET_IPPROTO_IP, ADR(pResult));
	(*SysSockParameter.parameterType := SysSocket2.SysSocket2_Type.STD;
	SysSockSpec.stdSockets.i32AddressFamily := SOCKET_AF_INET;
	SysSockSpec.stdSockets.i32Type := SOCKET_DGRAM;
	SysSockSpec.stdSockets.i32Protocol := SOCKET_IPPROTO_IP;
	SysSockParameter.specific := SysSockSpec;
	socket := SysSocket2.SysSock2Create(pParameter:= ADR(SysSockParameter), pResult:= ADR(pResult));*)	
	socket := SysSockCreate(SOCKET_AF_INET, SOCKET_DGRAM, SOCKET_IPPROTO_IP, ADR(pResult));
	IF socket < 0 THEN
		c_status := 1; (* SysSock2Create failed *)
		state := C_CLOSE;
	ELSE
		FunctionResult :=SysSockSetOption(socket, SOCKET_SOL, SOCKET_SO_BROADCAST, ADR(dint_true), SIZEOF(dint_true)); (* allow broadcast *)
		FunctionResult :=SysSockIoctl(socket, SOCKET_FIONBIO, ADR(dint_true)); (* put socket in non-blocking mode *)
		sockaddr.sin_family := SOCKET_AF_INET;
		sockaddr.sin_port := SysSockHtons(c_port);
		sockaddr.sin_addr.ulAddr := SEL(c_mode = 1, SOCKET_INADDR_ANY, SysSockNtohl(c_ip));

		IF c_mode >= 2 THEN (* SERVER Mode *)
			FunctionResult := SysSockBind(socket, ADR(sockaddr), SIZEOF(sockaddr));
			IF FunctionResult=0 THEN
				c_ready := TRUE; (* Connected *)
				state:= C_WAIT;
			ELSE
				c_status := 2; (* SysSock2Bind failed *)
				state := C_CLOSE;
			END_IF;
		ELSE
			c_ready := TRUE; (* Connected *)
			state:= C_WAIT;
		END_IF;
	END_IF;
	

(* ---------------------------------------------- *)

TC_INIT: (* TCP-CLIENT (AKTIV) *)
	// Create handle to ethernet socket to send messages
	//socket        := SysSock2Create(SOCKET_AF_INET, SOCKET_STREAM, SOCKET_IPPROTO_TCP, ADR(pResult)); 
	IF TLS THEN
		SysSockParameter.parameterType := SysSocket2.SysSocket2_Type.TLS;
		SysSockSpec.tlsSockets.hTlsContext := CmpTls.CmpTlsCreateContext(
			hCert:= RTS_INVALID_HANDLE, 
			tlsMethod:= TLS_CONFIG^.tlsMethod, 
			cipherList:= ADR(TLS_CONFIG^.chiperList),
			verifyMode := TLS_CONFIG^.verifyMode,
			pResult:= ADR(pResult));
			SysSockParameter.specific := SysSockSpec;	
	ELSE
		SysSockParameter.parameterType := SysSocket2.SysSocket2_Type.STD;
		SysSockSpec.stdSockets.i32AddressFamily := SOCKET_AF_INET;
		SysSockSpec.stdSockets.i32Type := SOCKET_STREAM;
		SysSockSpec.stdSockets.i32Protocol := SOCKET_IPPROTO_TCP;
		SysSockParameter.specific := SysSockSpec;	
	END_IF
	
	
	socket := SysSocket2.SysSock2Create(pParameter:= ADR(SysSockParameter), pResult:= ADR(pResult));	
	IF socket < 0 OR pResult <> CmpErrors.Errors.ERR_OK THEN
		c_status := 1;  (* SysSock2Create failed *)
		state := C_CLOSE;
	ELSE
		IF plc_841 OR plc_881 THEN
			FunctionResult :=SysSock2SetOption(socket,6,SOCKET_TCP_NODELAY, ADR(dint_true), SIZEOF(dint_true)); (* Set Push-Bit *)
		END_IF;
		// Set option for local address reuse
		FunctionResult :=SysSock2SetOption(socket, SOCKET_SOL, SOCKET_SO_REUSEADDR, ADR(dint_true), SIZEOF(dint_true));
		// Set option for keepalive
		//FunctionResult := SysSock2SetOption(socket, SOCKET_SOL, SOCKET_SO_KEEPALIVE, ADR(dint_true), SIZEOF(dint_true));
		IF TLS THEN
			FunctionResult :=SysSock2Ioctl(socket, SOCKET_FIONBIO, ADR(dint_false)); (* Blocking mode for connect to TLS*)
		ELSE
        	FunctionResult :=SysSock2Ioctl(socket, SOCKET_FIONBIO, ADR(dint_true)); (* NonBlocking mode *)
		END_IF
		sockaddr.sin_family := SOCKET_AF_INET;
		sockaddr.sin_port := SysSock2Ntohs(c_port);
		sockaddr.sin_addr.ulAddr  := SysSock2Ntohl(c_ip);
		c_select := FALSE;
		state := TC_CONNECT;
	END_IF;

(* ---------------------------------------------- *)

TC_CONNECT:
	IF NOT c_enable OR c_status = 255 THEN (* keine freigabe oder connect timeout *)
			state:= C_CLOSE;
	ELSE
		IF c_select = FALSE THEN
			TlsConnectLastTick := OSCAT_BASIC.T_PLC_MS();
			{info 'TODO: hind that this is blocking!'}
			pResult:=SysSock2Connect(socket,ADR(sockaddr),SIZEOF(sockaddr));
			TlsConnectTime := OSCAT_BASIC.T_PLC_MS() - TlsConnectLastTick; 
			IF pResult = CmpErrors.Errors.ERR_OK OR pResult =  CmpErrors.Errors.ERR_SOCK_ISCONNECTED THEN 
				c_ready := TRUE; (* Connected *)
				state:= C_WAIT;
				IF TLS THEN
        			SysSock2Ioctl(socket, SOCKET_FIONBIO, ADR(dint_true)); (* NonBlocking mode *)
				END_IF
			ELSE
				IF tls THEN
					state:= C_CLOSE;//TLS connect ist blokierend, wenn hier, fehler, reset 
				ELSE
					(* Connect durchgeführt, aber noch nicht verbunden, dann optional mit select-abfrage weitermachen *)
					c_select := SYSLIBSOCKETS_OPTION.0; (* Bit 0 = TCP-Client - use SysSock2select *)
				END_IF
				//c_select := TRUE;
			END_IF;

		
		ELSE
			c_Timeout.tv_sec := 0;
			c_Timeout.tv_usec := 0;
			c_fdWrite.fd_count := 1;
			c_fdWrite.fd_array[0] := socket;
			//IF SysSock2Select(SOCKET_FD_SETSIZE,0,ADR(c_fdWrite),0, ADR(c_Timeout), ADR(pResult)) > 0 THEN
			IF SysSocket2.SysSock2Select(
				hSocket:= socket, 
				diWidth:= SOCKET_FD_SETSIZE, 
				pfdRead:= 0, 
				pfdWrite:= ADR(c_fdWrite), 
				pfdExcept:= 0, 
				ptvTimeout:= ADR(c_Timeout), 
				pdiReady:= ADR(pResult)) > 0 THEN
				c_ready := TRUE; (* Connected *)
				state:= C_WAIT;
				IF TLS THEN
        			FunctionResult :=SysSock2Ioctl(socket, SOCKET_FIONBIO, ADR(dint_true)); (* NonBlocking mode *)
				END_IF
			END_IF;
		END_IF;
	END_IF;

(* ---------------------------------------------- *)

TS_INIT: (* TCP-SERVER (PASSIV) *)
	//	server_socket := SysSock2Create(SOCKET_AF_INET, SOCKET_STREAM, SOCKET_IPPROTO_IP, ADR(pResult)); (* Create Socket *)
	SysSockParameter.parameterType := SysSocket2.SysSocket2_Type.STD;
	SysSockSpec.stdSockets.i32AddressFamily := SOCKET_AF_INET;
	SysSockSpec.stdSockets.i32Type := SOCKET_STREAM;
	SysSockSpec.stdSockets.i32Protocol := SOCKET_IPPROTO_IP;
	SysSockParameter.specific := SysSockSpec;
	server_socket := SysSocket2.SysSock2Create(pParameter:= ADR(SysSockParameter), pResult:= ADR(pResult));
	
	IF server_socket = RTS_INVALID_HANDLE THEN
		c_status := 1; (* SysSock2Create failed *)
		state:= C_CLOSE;
	ELSE (* Address bindings *)
		SysSock2SetOption( server_socket, SOCKET_SOL, SOCKET_SO_REUSEADDR, ADR(dint_true), SIZEOF(dint_true) );
		sockaddr.sin_family:= SOCKET_AF_INET;
		sockaddr.sin_port := SysSock2Htons(c_port);
		sockaddr.sin_addr.ulAddr  := SOCKET_INADDR_ANY;
		IF NOT SysSock2Bind(server_socket, ADR(sockaddr), SIZEOF(sockaddr)) = 0 THEN
			c_status := 2; (* SysSock2Bind failed *)
			state := C_CLOSE;
		ELSIF NOT SysSock2Listen(server_socket, 1) = 0 THEN (* erzeugt Warteschlange für eine Verbindung *)
			c_status := 3; (* SysSock2Listen failed *)
			state:= C_CLOSE;
		ELSE
			SysSock2Ioctl(server_socket, SOCKET_FIONBIO, ADR(dint_true)); (* NonBlocking mode *)
			state:= TS_OPEN;
		END_IF;
	END_IF;

(* ---------------------------------------------- *)

TS_OPEN: (* Waiting for incomming connection *)
	sockaddr_size := SIZEOF(sockaddr);
	socket := SysSock2Accept(server_socket, ADR(sockaddr), ADR(sockaddr_size), ADR(pResult));

	IF socket <> RTS_INVALID_HANDLE THEN (* neuer Verbindungswunsch vorhanden *)
		IF c_mode = BYTE#2 AND sockaddr.sin_addr.ulAddr <> SysSock2Ntohl(c_ip) THEN (* Mode 2 = TCP + PASSIVE + PORT + IP  auf richtige Partner-IP prüfen *)
			state:= C_CLOSE;
		ELSE
			IF plc_841 OR plc_881 THEN
				SysSock2SetOption(socket, 6, SOCKET_TCP_NODELAY, ADR(dint_true), SIZEOF(dint_true)); (* Set Push-Bit *)
			END_IF;
			SysSock2Ioctl(socket, SOCKET_FIONBIO, ADR(dint_true)); (* NonBlocking mode *)
			c_ready := TRUE; (* Connected *)
			state := C_WAIT;
		END_IF;
	ELSIF NOT c_enable THEN (* keine freigabe mehr ? *)
			state:= C_CLOSE;
	END_IF;

(* ---------------------------------------------- *)

C_WAIT: (* Warten auf Anforderung für Beenden *)
	IF NOT c_enable OR NOT c_ready THEN
		state:= C_CLOSE;
	END_IF

(* ---------------------------------------------- *)

C_CLOSE: (* Close the Sockets *)
	c_ready := FALSE;
	IF socket >= 0 THEN
		IF (NOT plc_841) AND (NOT plc_881) THEN
			IF udp_mode THEN
				SysSockShutdown(socket, 0);
			ELSE
				SysSock2Shutdown(socket, 0); (* 870 *)
			END_IF
		END_IF;
		IF udp_mode THEN
			pResult := SysSockClose(socket);
		ELSE
			pResult := SysSock2Close(socket);	
		END_IF
		IF TLS THEN
			// cleanup TLS Context
			CmpTls.CmpTlsFreeContext(hTlsContext:= SysSockSpec.tlsSockets.hTlsContext);
		END_IF
		socket := RTS_INVALID_HANDLE;
		SysSockSpec.tlsSockets.hTlsContext := RTS_INVALID_HANDLE; 
	END_IF
	IF server_socket >= 0 THEN
		IF (NOT plc_841) AND (NOT plc_881) THEN
			SysSock2Shutdown(server_socket, 0); (* 870 *)
		END_IF;
		SysSock2Close(server_socket);
		server_socket := RTS_INVALID_HANDLE;
	END_IF
	state:= STOP;
END_CASE;

(* ---------------------------------------------- *)

IF c_ready THEN
	IF NOT c_ready_old THEN (* Verbindung aufgebaut - positive Flanke erkannt *)
		IP_C.C_STATE := 254;
		IP_C.TIME_RESET := TRUE; (* Alle Timer ruecksetzen *)
		(* ---------------------- Debug-Message ----------------------------*)
		(*IF _debug_enable THEN
			LOG_CL.NEW_MSG := 'IP_CON: CONNECTED -IP_ID ~6';
			LOG_CL.PRINTF[6] := INT_TO_STRING(debug_ID);
			LOG_MSG();
		END_IF;*)
		(* -----------------------------------------------------------------------------*)
	ELSE
		IP_C.C_STATE := 255; (* Verbindung ist aufgebaut *)
	END_IF;
ELSE
	IF c_ready_old THEN (* Verbindung abgebaut - negative Flanke erkannt *)
		IP_C.C_STATE := 1;
		IP_C.MAILBOX[1] := 0; (* Receive Info rücksetzen *)
		IP_C.MAILBOX[2] := 0; (* Send-Pause rücksetzen *)
		IP_C.MAILBOX[3] := 0; (* Receive-Pause rücksetzen *)
		IF NOT new_connection THEN
			s_active := FALSE; (* Sendeaktivitäten stoppen *)
			s_req := FALSE; (* Sendefreigabe rücksetzen *)
			S_BUF.SIZE := 0; (* Sendelänge löschen *)
			(*IP_C.TIME_RESET := TRUE;*) (* Alle Timer ruecksetzen *)
		END_IF;
		(* ---------------------- Debug-Message ----------------------------*)
		(*IF _debug_enable THEN
			LOG_CL.NEW_MSG := 'IP_CON: DISCONNECTED';
			LOG_MSG();
		END_IF;*)
		(* -----------------------------------------------------------------------------*)
	ELSE
		IP_C.C_STATE := 0; (* Verbindung ist abgebaut *)
	END_IF;
END_IF;

c_ready_old := c_ready;

(* Der Datenempfang wird angehalten solange ein Sendevorgang läuft *)
(* sonst kann es vorkommen das die Antwort-daten schon empfangen werden, *)
(* bevor der Sendevorgang vom programm abgeschlossen wurde *)

IF c_ready AND NOT s_active AND IP_C.MAILBOX[3] = 0 THEN
	IF R_BUF.SIZE >= INT_TO_UINT(r_max_size) THEN
		R_BUF.SIZE := UINT#0;
		r_status := 254; (* Empfangsbuffer wegen Überlauf rückgesetzt *)
	END_IF;

	r_offset := SEL(udp_mode,UINT_TO_INT(R_BUF.SIZE),0);
	r_count := r_max_size - r_offset;

	IF udp_mode THEN
		//bytes_received := SysSock2RecvFrom(socket, ADR(R_BUF.BUFFER), r_count, 0, ADR(sockaddr), SIZEOF(sockaddr), ADR(pResult));
		(*bytes_received := SysSock2RecvFrom(
	hSocket:= socket, 
	pbyBuffer:= ADR(R_BUF.BUFFER), 
	diBufferSize:= r_count, 
	diFlags:= 0, 
	pSockAddr:= ADR(sockaddr), 
	diSockAddrSize:= SIZEOF(sockaddr), 
	pResult:= ADR(pResult));*)
	bytes_received := TO_DINT(SysSockRecvFrom(socket, ADR(R_BUF.BUFFER), r_count, 0, ADR(sockaddr), SIZEOF(sockaddr), ADR(pResult)));
		IF c_mode = BYTE#3 AND sockaddr.sin_addr.ulAddr <> SysSockNtohl(c_ip) THEN (* Mode 3 = UDP + PASSIVE + PORT + IP  auf richtige Partner-IP prüfen *)
			bytes_received := 0;
			R_BUF.SIZE := UINT#0;
			sockaddr.sin_port := SysSockNtohs(c_port);
			sockaddr.sin_addr.ulAddr  := SysSockNtohl(c_ip);
		END_IF;

	ELSE
		bytes_received := TO_DINT(SysSock2Recv(socket, ADR(R_BUF.BUFFER[r_offset]), r_count, 0, ADR(pResult)));
	END_IF;

	CASE pResult OF
		518:  bytes_received:=-1; //Connection OKAY just no data and do not want to BIND
		521:  bytes_received:=0; //Connection has been refused by the remote host 
		523:  bytes_received:=0; //The host has not been found  
		524:  bytes_received:=0; //Host is unreachable  
		526:  bytes_received:=0; //The socket is not connected  
		527:  bytes_received:=0; //Shutdown has been called on the socket  
		529:  bytes_received:=0; //Socket has been gracefully closed. No more send/receives allowed	 
	END_CASE

	
	(*UDP: IPC returns -1 if no data available or error occured,841 returns -1 if error occured and 0 if no data available*)
	CASE bytes_received OF
	-2147483648..-1: ; (* No data available or error occured *)
	 0: IF NOT udp_mode OR pResult<>518 THEN (* TCP-Mode: socket wurde von remote geschlossen *)
			c_status := 253;
			c_ready := FALSE;
		END_IF;
	ELSE (* daten wurden empfangen *)
  		r_time := tx; (* Receive Timer ruecksetzen *)
		R_BUF.SIZE := INT_TO_UINT(r_offset) + DINT_TO_UINT(bytes_received); (* aktuelle buffersize eintragen *)
		IP_C.MAILBOX[1] := IP_C.MAILBOX[1] + 1; (* Receive Info *)
		IF IP_C.MAILBOX[1] = 0 THEN IP_C.MAILBOX[1] := 1; END_IF;

		(* ---------------------- Debug-Message ----------------------------*)
		(*IF _debug_enable THEN
			LOG_CL.NEW_MSG := 'IP_REC DATA: POS: ~1 : SIZE: ~2 TOTAL ~3 -IP_ID ~6';
			LOG_CL.PRINTF[1] := INT_TO_STRING(r_offset);
			LOG_CL.PRINTF[2] := INT_TO_STRING(r_count);
			LOG_CL.PRINTF[3] := UINT_TO_STRING(R_BUF.SIZE);
			LOG_CL.PRINTF[6] := INT_TO_STRING(debug_ID);
			LOG_MSG();
		END_IF;*)
		(* -----------------------------------------------------------------------------*)

	END_CASE
END_IF;

(* ---------------------------------------------- *)

IF S_BUF.SIZE > 0 THEN
	IF c_ready AND c_enable THEN
		IF NOT s_active AND IP_C.MAILBOX[2] = 0 THEN
			(* Gesamtanzahl an Bytes limitieren und uebergeben *)
			s_total := LIMIT(0,UINT_TO_INT(S_BUF.SIZE),r_max_size);
			s_cur_pos  := 0;
			s_cur_size := 0;
			s_start := TRUE; (* Daten kopieren und senden anstossen *)
			s_active := TRUE; (* Sende-Betrieb aktivieren *)
			(* ---------------------- Debug-Message ----------------------------*)
			(*IF _debug_enable THEN
				LOG_CL.NEW_MSG := 'IP_SEN INIT: TOTAL: ~1 -IP_ID ~6';
				LOG_CL.PRINTF[1] := INT_TO_STRING(S_TOTAL);
				LOG_CL.PRINTF[6] := INT_TO_STRING(debug_ID);
				LOG_MSG();
			END_IF;*)
			(* -----------------------------------------------------------------------------*)
		END_IF;

		IF s_done OR s_start THEN (* Daten senden aktiv *)

			s_start := FALSE;
			s_cur_pos := s_cur_pos + s_cur_size; (* neue Sende-Datenposition bestimmen *)
			IF s_total > s_cur_pos THEN (* weitere Daten zum senden vorhanden ? *)
				s_cur_size := s_total - s_cur_pos;
				s_cur_size := LIMIT(0, s_cur_size, s_max_size); (* Telegrammlänge begrenzen *)
				(* ---------------------- Debug-Message ----------------------------*)
				(*IF _debug_enable THEN
					LOG_CL.NEW_MSG := 'IP_SEN DATA: POS: ~1 : SIZE: ~2 TOTAL ~3 -IP_ID ~6';
					LOG_CL.PRINTF[1] := INT_TO_STRING(S_CUR_POS);
					LOG_CL.PRINTF[2] := INT_TO_STRING(S_CUR_SIZE);
					LOG_CL.PRINTF[3] := INT_TO_STRING(S_TOTAL);
					LOG_CL.PRINTF[6] := INT_TO_STRING(debug_ID);
					LOG_MSG();
				END_IF;*)
				(* -----------------------------------------------------------------------------*)
				s_time := tx; (* Send Timer ruecksetzen *)
				r_time := tx; (* Receive Timer ruecksetzen *)
				s_req := TRUE;

			ELSE
				(* keine weitere Sendedaten vorhanden -> Senden beenden *)
				s_req := FALSE;
				s_active := FALSE;
				S_BUF.SIZE := 0;
				(* ---------------------- Debug-Message ----------------------------*)
				(*IF _debug_enable THEN
					LOG_CL.NEW_MSG := 'IP_SEN FINISH -IP_ID ~6';
					LOG_CL.PRINTF[6] := INT_TO_STRING(debug_ID);
					LOG_MSG();
				END_IF;*)
				(* -----------------------------------------------------------------------------*)
			END_IF;
		END_IF;
	END_IF;
END_IF;

IF s_req THEN
	s_done := FALSE;
	IF udp_mode THEN
		bytes_sent := TO_DINT(SysSockSendTo(socket, ADR(S_BUF.BUFFER[s_cur_pos]), s_cur_size, 0, ADR(sockaddr), SIZEOF(sockaddr), ADR(pResult)));
	ELSE
		bytes_sent := TO_DINT(SysSock2Send(socket, ADR(S_BUF.BUFFER[s_cur_pos]), s_cur_size, 0, ADR(pResult)));
	END_IF;

	CASE bytes_sent OF
	-2147483648..-1:	; (* ERROR: Noch nicht bereit um Daten aufzunehmen -> nächsten Zyklus wieder probieren *)
	 0: IF NOT udp_mode THEN (* TCP-Mode: socket wurde von remote geschlossen *)
			c_status := 253;
			c_ready := FALSE;
		END_IF;
	ELSE
		s_done := TRUE;
		s_cur_size := DINT_TO_INT(bytes_sent); (* Anzahl der wirklich versendeten Bytes übernehmen *)
		(* ---------------------- Debug-Message ----------------------------*)
		(*IF _debug_enable THEN
			LOG_CL.NEW_MSG := 'IP_SEN SEND_COUNT ~1 -IP_ID ~6';
			LOG_CL.PRINTF[1] := DINT_TO_STRING(s_cur_size);
			LOG_CL.PRINTF[6] := INT_TO_STRING(debug_ID);
			LOG_MSG();
		END_IF;*)
		(* -----------------------------------------------------------------------------*)
	END_CASE
END_IF;

(* ---------------------------------------------- *)

IF IP_C.R_OBSERVE = FALSE OR s_active THEN
    r_time := tx;
END_IF;

IF c_status = 0 AND tx - c_time > error_time AND c_enable AND NOT c_ready AND c_mode < 2 THEN (* Connect Timeout *)
	c_status := 255; (* Timeout-Fehler ausgeben *)
END_IF;
IF s_status = 0 AND tx - s_time > error_time AND s_active THEN (* Send Timeout *)
	s_status := 255; (* Timeout-Fehler ausgeben *)
END_IF;
IF r_status = 0 AND tx - r_time > error_time AND c_ready AND IP_C.R_OBSERVE THEN (* Receive Timeout *)
	r_status := 255; (* Timeout-Fehler ausgeben *)
END_IF;

IP_C.ERROR := OSCAT_BASIC.DWORD_OF_BYTE(c_status,s_status,r_status,0);

(* ---------------------- Debug-Message ----------------------------*)
(*IF  _debug_enable THEN
	IF (IP_C.ERROR <> debug_lasterror) THEN
		LOG_CL.NEW_MSG := 'IP_ERROR ~1 -IP_ID ~6';
		LOG_CL.PRINTF[1] := DWORD_TO_STRING(IP_C.ERROR);
		LOG_CL.PRINTF[6] := INT_TO_STRING(debug_ID);
		LOG_MSG();

		debug_lasterror := IP_C.ERROR;
		debug_last_id := debug_ID;
	END_IF;
END_IF;*)
(* -----------------------------------------------------------------------------*)

(* revision history
ks	18. oct. 2008	rev 1.0
	original version
ks	05. jan. 2009	rev 1.1
	zusätzlichen Parameter "Port" hinzugefügt, und Code bei Verbindungsaufbau angepasst
ks	28. feb. 2009	rev 1.2
	connect code angepasst und verkürzung der zyklen bei Send
ks	20. oct. 2009	rev 1.3
	network_buffer basis 0
ks	06. dec. 2009	rev 1.4
	receive_count MAILBOX[1]
ks	10. nov. 2010	rev 1.5
	send_pause MAILBOX[2] and receive_pause MAILBOX[3] 
ks	07. feb. 2011	rev 1.6
	Fehlercode 253 bei Remote-Verbindungsabbruch
ks	30. may. 2011	rev 1.7
	Fehler bei Empfangsüberwachung
ks	26. july. 2011	rev 1.8
	Error-Reset, diverse optimierungen 
ks	26. feb. 2012	rev 1.9
	Code-Optimierung für höhere kompatibilität

*)

END_FUNCTION_BLOCK

// Common/Function Blocks/IP_CONTROL_135
FUNCTION_BLOCK IP_CONTROL_135

VAR_IN_OUT
	IP_C : IP_C; (* IP_Control Verwaltungsstruktur *)
	S_BUF : NETWORK_BUFFER; (* Externer Sendbuffer *)
	R_BUF : NETWORK_BUFFER; (* Externer Receivebuffer *)
END_VAR
VAR_INPUT
	IP : DWORD; (* IP Adresse *)
	PORT : WORD; (* Port Nummer *)
	TIME_OUT : TIME; (* Ueberwachungszeit Connect / Send / Receive *)
END_VAR
VAR
	c_time : UDINT; (* CONNECT-Time (Zeit bei nicht vorhandener Verbindung) *)
	s_time : UDINT; (* SEND-Time    (Zeit seit letzten Datensenden) *)
	r_time : UDINT; (* RECEIVE-Time (Zeit seit letztem Datenempfang) *)

	c_enable : BOOL; (* Connect: freigabe *)
	c_ip : DWORD; (* Connect: aktuelle IP-Adresse *)
	c_port : WORD; (* Connect: aktuelle Port-Nummer *)
	c_mode : BYTE; (* Connect: aktueller Mode UDP/TCP...... *)
	c_status : BYTE; (* Connect: Status (Errorcode) *)
	c_ready : BOOL; (* Connect: Verbindung aufgebaut *)
	c_ready_old : BOOL; (* Connect: letzter Zustand von c_ready für Flankenauswertung *)
	c_select : BOOL; (* non blocking mode - abfrage über select durchführen *)
	c_fdWrite : SOCKET_FD_SET;
	c_Timeout : SOCKET_TIMEVAL;

	s_total : INT; (* Send: Gesamtanzahl Bytes zum senden *)
	s_cur_pos : INT; (* Send: aktuelle Sendeposition *)
	s_cur_size : INT; (* Send: aktuelle Sendegroesse *)
	s_max_size : INT; (* Send: maximale Telegrammlänge fuer Senden *)
	s_start : BOOL; (* Send: Sende modus aktivieren *)
	s_active : BOOL; (* Send: Daten senden ist aktiv *)
	s_req : BOOL; (* Send: Start Daten senden *)
	s_done : BOOL; (* Send: ohne Fehler beendet *)
	s_status : BYTE; (* Send: Status (Errorcodes) *)

	r_status : BYTE; (* Receive: Status (Errorcodes) *)
	r_count : INT; (* Receive: Anzahl empfangener Bytes *)
	r_offset : INT; (* Receive: aktuelle Position in externen Receivebuffer *)
	r_max_size : INT; (* Receive: groesse des externen Empfangbuffers*)

	new_connection : BOOL; (* Neue Verbindungsparameter vorhanden *)
	tx : DWORD; (* letzter zeitwert *)
	error_time : DWORD; (* aktueller Timeout-Wert *)

	state: BYTE; (* schrittmerker für connect *)
	server_socket : RTS_IEC_HANDLE:= RTS_INVALID_HANDLE; 
	socket : RTS_IEC_HANDLE:= RTS_INVALID_HANDLE;
	sockaddr : SOCKADDRESS;
	sockaddr_size : DWORD;
	plc_841 : BOOL;
	plc_881 : BOOL;
	dint_true : DINT := 1;
	bytes_received : DINT;
	bytes_sent : DINT;
	udp_mode : BOOL;
	pResult : UDINT; //Needed for V3 Lib
	(*LOG_MSG : LOG_MSG;
	_debug_enable : BOOL := TRUE;
	debug_index : INT;
	debug_ID : INT;
	debug_lasterror : DWORD;
	debug_last_id : INT := 255;
	state_last: BYTE;*)

END_VAR

VAR CONSTANT
	STOP : BYTE := 0;
	TS_INIT: BYTE := 1;
	TS_OPEN : BYTE:= 2;

	UDP_INIT : BYTE:= 31;

	TC_INIT : BYTE:= 51;
	TC_CONNECT : BYTE:= 52;

	C_WAIT : BYTE:= 250;
	C_CLOSE : BYTE:= 251;

END_VAR

(*

version 1.9		26. Feb. 2012
programmer 		ks
tested by			ks

IP_CONTROL ist ein Wrapper-Baustein um eine Hersteller neutrale Schnittstelle zum Ethernet zu schaffen
*)

(* ---------------------- Debug-Message ----------------------------*)
(*IF _debug_enable THEN
	IF IP_C.FIFO.ID > BYTE#0 THEN
		debug_index := IP_C.FIFO.NR;
		debug_ID := BYTE_TO_INT(IP_C.FIFO.X[debug_index]);
	END_IF;
END_IF;*)
(* -----------------------------------------------------------------------------*)

(* read system time *)
tx := OSCAT_BASIC.T_PLC_MS();

IF IP_C.C_PORT = 0 THEN
	IP_C.C_PORT := PORT; (* uebergebenen PORT durch parametrierten PORT ersetzen *)
END_IF;
IF IP_C.C_IP = 0 AND IP_C.C_MODE < 4 THEN
	IP_C.C_IP := IP; (* uebergebene IP durch paramtrierte IP ersetzen *)
END_IF;

new_connection := c_ip <> IP_C.C_IP OR c_mode <> IP_C.C_MODE OR c_port <> IP_C.C_PORT; (* neue Verbindungs erwünscht ? *)
c_enable := IP_C.C_ENABLE AND NOT new_connection;

IF IP_C.C_ENABLE AND IP_C.ERROR = 0 AND state = STOP THEN (* Freigabe,kein Fehler,kein Socket offen *)
	c_ip   := IP_C.C_IP;
	c_mode := IP_C.C_MODE;
	c_port := IP_C.C_PORT;
	plc_841 := SYSLIBSOCKETS_OPTION.1; (* Bit 1 = WAGO 750-841 *)
	plc_881 := SYSLIBSOCKETS_OPTION.2; (* Bit 1 = WAGO 750-881 *)
	udp_mode := C_MODE.0; (* Mode 1,3,5 = udp *)

	error_time := TIME_TO_DWORD(MAX(T#200ms,TIME_OUT));
	IP_C.TIME_RESET := TRUE; (* Alle Timer ruecksetzen *)

	r_max_size := SIZEOF(R_BUF.BUFFER);
	s_max_size := SIZEOF(S_BUF.BUFFER);

	IF C_MODE.0 THEN (* Mode: 1,3,5 = UDP CLIENT/SERVER *)
		state := UDP_INIT;
	ELSIF C_MODE = 0 THEN (* Mode: 0 = TCP CLIENT *)
		state := TC_INIT;
	ELSE
		state := TS_INIT; (* Mode: 2,4 = TCP SERVER *)
	END_IF;

	(* ---------------------- Debug-Message ----------------------------*)
	(*IF _debug_enable THEN
		LOG_CL.NEW_MSG := 'IP_CON: MODE ~1 / IP ~2 / PORT ~3 /ID ~6';
		LOG_CL.PRINTF[1] := BYTE_TO_STRING(C_MODE);
		LOG_CL.PRINTF[2] := IP4_TO_STRING(c_ip);
		LOG_CL.PRINTF[3] := WORD_TO_STRING(c_port);
		LOG_CL.PRINTF[6] := INT_TO_STRING(debug_ID);
		LOG_MSG();
	END_IF;*)
	(* -----------------------------------------------------------------------------*)

END_IF;

(* ---------------------- Debug-Message ----------------------------*)
(*IF  _debug_enable THEN
	IF state <> state_last THEN
		LOG_CL.NEW_MSG := 'IP_STEP ~1 -IP_ID ~6';
		LOG_CL.PRINTF[1] := BYTE_TO_STRING(state);
		LOG_CL.PRINTF[6] := INT_TO_STRING(debug_ID);
		LOG_MSG();
		state_last := state;
	END_IF;
END_IF;*)
(* -----------------------------------------------------------------------------*)

IF IP_C.TIME_RESET THEN (* Alle Timer ruecksetzen *)
	IP_C.TIME_RESET := FALSE; (* Reset rücksetzen *)
	c_time := tx; (* Connect Timer ruecksetzen *)
	s_time := tx; (* Send Timer ruecksetzen *)
	r_time := tx; (* Receive Timer ruecksetzen *)

	c_status := BYTE#0; (* letzten Connect Fehler rücksetzen *)
	s_status := BYTE#0; (* letzten Send Fehler rücksetzen *)
	r_status := BYTE#0; (* letzten Receive Fehler rücksetzen *)
END_IF;

(* ---------------------------------------------- *)

CASE state OF

UDP_INIT: (* UDP_CLIENT + SERVER *)
	socket := SysSockCreate(SOCKET_AF_INET, SOCKET_DGRAM, SOCKET_IPPROTO_IP, ADR(pResult));
	IF socket < 0 THEN
		c_status := 1; (* SysSockCreate failed *)
		state := C_CLOSE;
	ELSE
		SysSockSetOption(socket, SOCKET_SOL, SOCKET_SO_BROADCAST, ADR(dint_true), SIZEOF(dint_true)); (* allow broadcast *)
		SysSockIoctl(socket, SOCKET_FIONBIO, ADR(dint_true)); (* put socket in non-blocking mode *)
		sockaddr.sin_family := SOCKET_AF_INET;
		sockaddr.sin_port := SysSockHtons(c_port);
		sockaddr.sin_addr.ulAddr := SEL(c_mode = 1, SOCKET_INADDR_ANY, SysSockNtohl(c_ip));

		IF c_mode >= 2 THEN (* SERVER Mode *)
			IF SysSockBind(socket, ADR(sockaddr), SIZEOF(sockaddr)) = 0 THEN
				c_ready := TRUE; (* Connected *)
				state:= C_WAIT;
			ELSE
				c_status := 2; (* SysSockBind failed *)
				state := C_CLOSE;
			END_IF;
		ELSE
			c_ready := TRUE; (* Connected *)
			state:= C_WAIT;
		END_IF;
	END_IF;

(* ---------------------------------------------- *)

TC_INIT: (* TCP-CLIENT (AKTIV) *)
	socket := SysSockCreate(SOCKET_AF_INET, SOCKET_STREAM, SOCKET_IPPROTO_IP, ADR(pResult));
	IF socket < 0 THEN
		c_status := 1;  (* SysSockCreate failed *)
		state := C_CLOSE;
	ELSE
		IF plc_841 OR plc_881 THEN
			SysSockSetOption(socket,6,SOCKET_TCP_NODELAY, ADR(dint_true), SIZEOF(dint_true)); (* Set Push-Bit *)
		END_IF;
		SysSockIoctl(socket, SOCKET_FIONBIO, ADR(dint_true)); (* NonBlocking mode *)
		sockaddr.sin_family := SOCKET_AF_INET;
		sockaddr.sin_port := SysSockNtohs(c_port);
		sockaddr.sin_addr.ulAddr := SysSockNtohl(c_ip);
		c_select := FALSE;
		state := TC_CONNECT;
	END_IF;

(* ---------------------------------------------- *)

TC_CONNECT:
	IF NOT c_enable OR c_status = 255 THEN (* keine freigabe oder connect timeout *)
			state:= C_CLOSE;
	ELSE
		IF c_select = FALSE THEN
			IF SysSockConnect(socket,ADR(sockaddr),SIZEOF(sockaddr)) = 0 THEN
				c_ready := TRUE; (* Connected *)
				state:= C_WAIT;
			ELSE
				(* Connect durchgeführt, aber noch nicht verbunden, dann optional mit select-abfrage weitermachen *)
				c_select := SYSLIBSOCKETS_OPTION.0; (* Bit 0 = TCP-Client - use SysSockselect *)
			END_IF;
		ELSE
			c_Timeout.tv_sec := 0;
			c_Timeout.tv_usec := 0;
			c_fdWrite.fd_count := 1;
			c_fdWrite.fd_array[0] := socket;
			IF SysSockSelect(SOCKET_FD_SETSIZE,0,ADR(c_fdWrite),0, ADR(c_Timeout), ADR(pResult)) > 0 THEN
				c_ready := TRUE; (* Connected *)
				state:= C_WAIT;
			END_IF;
		END_IF;
	END_IF;

(* ---------------------------------------------- *)

TS_INIT: (* TCP-SERVER (PASSIV) *)
	server_socket := SysSockCreate(SOCKET_AF_INET, SOCKET_STREAM, SOCKET_IPPROTO_IP, ADR(pResult)); (* Create Socket *)
	IF server_socket = RTS_INVALID_HANDLE THEN
		c_status := 1; (* SysSockCreate failed *)
		state:= C_CLOSE;
	ELSE (* Address bindings *)
		SysSockSetOption( server_socket, SOCKET_SOL, SOCKET_SO_REUSEADDR, ADR(dint_true), SIZEOF(dint_true) );
		sockaddr.sin_family:= SOCKET_AF_INET;
		sockaddr.sin_port := SysSockHtons(c_port);
		sockaddr.sin_addr.ulAddr := SOCKET_INADDR_ANY;
		IF NOT SysSockBind(server_socket, ADR(sockaddr), SIZEOF(sockaddr)) = 0 THEN
			c_status := 2; (* SysSockBind failed *)
			state := C_CLOSE;
		ELSIF NOT SysSockListen(server_socket, 1) = 0 THEN (* erzeugt Warteschlange für eine Verbindung *)
			c_status := 3; (* SysSockListen failed *)
			state:= C_CLOSE;
		ELSE
			SysSockIoctl(server_socket, SOCKET_FIONBIO, ADR(dint_true)); (* NonBlocking mode *)
			state:= TS_OPEN;
		END_IF;
	END_IF;

(* ---------------------------------------------- *)

TS_OPEN: (* Waiting for incomming connection *)
	sockaddr_size := SIZEOF(sockaddr);
	socket := SysSockAccept(server_socket, ADR(sockaddr), ADR(sockaddr_size), ADR(pResult));

	IF socket <> RTS_INVALID_HANDLE THEN (* neuer Verbindungswunsch vorhanden *)
		IF c_mode = BYTE#2 AND sockaddr.sin_addr.ulAddr <> SysSockNtohl(c_ip) THEN (* Mode 2 = TCP + PASSIVE + PORT + IP  auf richtige Partner-IP prüfen *)
			state:= C_CLOSE;
		ELSE
			IF plc_841 OR plc_881 THEN
				SysSockSetOption(socket, 6, SOCKET_TCP_NODELAY, ADR(dint_true), SIZEOF(dint_true)); (* Set Push-Bit *)
			END_IF;
			SysSockIoctl(socket, SOCKET_FIONBIO, ADR(dint_true)); (* NonBlocking mode *)
			c_ready := TRUE; (* Connected *)
			state := C_WAIT;
		END_IF;
	ELSIF NOT c_enable THEN (* keine freigabe mehr ? *)
			state:= C_CLOSE;
	END_IF;

(* ---------------------------------------------- *)

C_WAIT: (* Warten auf Anforderung für Beenden *)
	IF NOT c_enable OR NOT c_ready THEN
		state:= C_CLOSE;
	END_IF

(* ---------------------------------------------- *)

C_CLOSE: (* Close the Sockets *)
	c_ready := FALSE;
	IF socket >= 0 THEN
		IF (NOT plc_841) AND (NOT plc_881) THEN
			SysSockShutdown(socket, 0); (* 870 *)
		END_IF;
		SysSockClose(socket);
		socket := RTS_INVALID_HANDLE;
	END_IF
	IF server_socket >= 0 THEN
		IF (NOT plc_841) AND (NOT plc_881) THEN
			SysSockShutdown(server_socket, 0); (* 870 *)
		END_IF;
		SysSockClose(server_socket);
		server_socket := RTS_INVALID_HANDLE;
	END_IF
	state:= STOP;
END_CASE;

(* ---------------------------------------------- *)

IF c_ready THEN
	IF NOT c_ready_old THEN (* Verbindung aufgebaut - positive Flanke erkannt *)
		IP_C.C_STATE := 254;
		IP_C.TIME_RESET := TRUE; (* Alle Timer ruecksetzen *)
		(* ---------------------- Debug-Message ----------------------------*)
		(*IF _debug_enable THEN
			LOG_CL.NEW_MSG := 'IP_CON: CONNECTED -IP_ID ~6';
			LOG_CL.PRINTF[6] := INT_TO_STRING(debug_ID);
			LOG_MSG();
		END_IF;*)
		(* -----------------------------------------------------------------------------*)
	ELSE
		IP_C.C_STATE := 255; (* Verbindung ist aufgebaut *)
	END_IF;
ELSE
	IF c_ready_old THEN (* Verbindung abgebaut - negative Flanke erkannt *)
		IP_C.C_STATE := 1;
		IP_C.MAILBOX[1] := 0; (* Receive Info rücksetzen *)
		IP_C.MAILBOX[2] := 0; (* Send-Pause rücksetzen *)
		IP_C.MAILBOX[3] := 0; (* Receive-Pause rücksetzen *)
		IF NOT new_connection THEN
			s_active := FALSE; (* Sendeaktivitäten stoppen *)
			s_req := FALSE; (* Sendefreigabe rücksetzen *)
			S_BUF.SIZE := 0; (* Sendelänge löschen *)
			(*IP_C.TIME_RESET := TRUE;*) (* Alle Timer ruecksetzen *)
		END_IF;
		(* ---------------------- Debug-Message ----------------------------*)
		(*IF _debug_enable THEN
			LOG_CL.NEW_MSG := 'IP_CON: DISCONNECTED';
			LOG_MSG();
		END_IF;*)
		(* -----------------------------------------------------------------------------*)
	ELSE
		IP_C.C_STATE := 0; (* Verbindung ist abgebaut *)
	END_IF;
END_IF;

c_ready_old := c_ready;

(* Der Datenempfang wird angehalten solange ein Sendevorgang läuft *)
(* sonst kann es vorkommen das die Antwort-daten schon empfangen werden, *)
(* bevor der Sendevorgang vom programm abgeschlossen wurde *)

IF c_ready AND NOT s_active AND IP_C.MAILBOX[3] = 0 THEN
	IF R_BUF.SIZE >= INT_TO_UINT(r_max_size) THEN
		R_BUF.SIZE := UINT#0;
		r_status := 254; (* Empfangsbuffer wegen Überlauf rückgesetzt *)
	END_IF;

	r_offset := SEL(udp_mode,UINT_TO_INT(R_BUF.SIZE),0);
	r_count := r_max_size - r_offset;

	IF udp_mode THEN
		bytes_received := SysSockRecvFrom(socket, ADR(R_BUF.BUFFER), r_count, 0, ADR(sockaddr), SIZEOF(sockaddr), ADR(pResult));

		IF c_mode = BYTE#3 AND sockaddr.sin_addr.ulAddr <> SysSockNtohl(c_ip) THEN (* Mode 3 = UDP + PASSIVE + PORT + IP  auf richtige Partner-IP prüfen *)
			bytes_received := 0;
			R_BUF.SIZE := UINT#0;
			sockaddr.sin_port := SysSockNtohs(c_port);
			sockaddr.sin_addr.ulAddr := SysSockNtohl(c_ip);
		END_IF;

	ELSE
		bytes_received := SysSockRecv(socket, ADR(R_BUF.BUFFER[r_offset]), r_count, 0, ADR(pResult));
	END_IF;

	(*UDP: IPC returns -1 if no data available or error occured,841 returns -1 if error occured and 0 if no data available*)
	CASE bytes_received OF
	-2147483648..-1: ; (* No data available or error occured *)
	 0: IF NOT udp_mode THEN (* TCP-Mode: socket wurde von remote geschlossen *)
			c_status := 253;
			c_ready := FALSE;
		END_IF;
	ELSE (* daten wurden empfangen *)
  		r_time := tx; (* Receive Timer ruecksetzen *)
		R_BUF.SIZE := INT_TO_UINT(r_offset + DINT_TO_UINT(bytes_received)); (* aktuelle buffersize eintragen *)
		IP_C.MAILBOX[1] := IP_C.MAILBOX[1] + 1; (* Receive Info *)
		IF IP_C.MAILBOX[1] = 0 THEN IP_C.MAILBOX[1] := 1; END_IF;

		(* ---------------------- Debug-Message ----------------------------*)
		(*IF _debug_enable THEN
			LOG_CL.NEW_MSG := 'IP_REC DATA: POS: ~1 : SIZE: ~2 TOTAL ~3 -IP_ID ~6';
			LOG_CL.PRINTF[1] := INT_TO_STRING(r_offset);
			LOG_CL.PRINTF[2] := INT_TO_STRING(r_count);
			LOG_CL.PRINTF[3] := UINT_TO_STRING(R_BUF.SIZE);
			LOG_CL.PRINTF[6] := INT_TO_STRING(debug_ID);
			LOG_MSG();
		END_IF;*)
		(* -----------------------------------------------------------------------------*)

	END_CASE
END_IF;

(* ---------------------------------------------- *)

IF S_BUF.SIZE > 0 THEN
	IF c_ready AND c_enable THEN
		IF NOT s_active AND IP_C.MAILBOX[2] = 0 THEN
			(* Gesamtanzahl an Bytes limitieren und uebergeben *)
			s_total := LIMIT(0,UINT_TO_INT(S_BUF.SIZE),r_max_size);
			s_cur_pos  := 0;
			s_cur_size := 0;
			s_start := TRUE; (* Daten kopieren und senden anstossen *)
			s_active := TRUE; (* Sende-Betrieb aktivieren *)
			(* ---------------------- Debug-Message ----------------------------*)
			(*IF _debug_enable THEN
				LOG_CL.NEW_MSG := 'IP_SEN INIT: TOTAL: ~1 -IP_ID ~6';
				LOG_CL.PRINTF[1] := INT_TO_STRING(S_TOTAL);
				LOG_CL.PRINTF[6] := INT_TO_STRING(debug_ID);
				LOG_MSG();
			END_IF;*)
			(* -----------------------------------------------------------------------------*)
		END_IF;

		IF s_done OR s_start THEN (* Daten senden aktiv *)

			s_start := FALSE;
			s_cur_pos := s_cur_pos + s_cur_size; (* neue Sende-Datenposition bestimmen *)
			IF s_total > s_cur_pos THEN (* weitere Daten zum senden vorhanden ? *)
				s_cur_size := s_total - s_cur_pos;
				s_cur_size := LIMIT(0, s_cur_size, s_max_size); (* Telegrammlänge begrenzen *)
				(* ---------------------- Debug-Message ----------------------------*)
				(*IF _debug_enable THEN
					LOG_CL.NEW_MSG := 'IP_SEN DATA: POS: ~1 : SIZE: ~2 TOTAL ~3 -IP_ID ~6';
					LOG_CL.PRINTF[1] := INT_TO_STRING(S_CUR_POS);
					LOG_CL.PRINTF[2] := INT_TO_STRING(S_CUR_SIZE);
					LOG_CL.PRINTF[3] := INT_TO_STRING(S_TOTAL);
					LOG_CL.PRINTF[6] := INT_TO_STRING(debug_ID);
					LOG_MSG();
				END_IF;*)
				(* -----------------------------------------------------------------------------*)
				s_time := tx; (* Send Timer ruecksetzen *)
				r_time := tx; (* Receive Timer ruecksetzen *)
				s_req := TRUE;

			ELSE
				(* keine weitere Sendedaten vorhanden -> Senden beenden *)
				s_req := FALSE;
				s_active := FALSE;
				S_BUF.SIZE := 0;
				(* ---------------------- Debug-Message ----------------------------*)
				(*IF _debug_enable THEN
					LOG_CL.NEW_MSG := 'IP_SEN FINISH -IP_ID ~6';
					LOG_CL.PRINTF[6] := INT_TO_STRING(debug_ID);
					LOG_MSG();
				END_IF;*)
				(* -----------------------------------------------------------------------------*)
			END_IF;
		END_IF;
	END_IF;
END_IF;

IF s_req THEN
	s_done := FALSE;
	IF udp_mode THEN
		bytes_sent := SysSockSendTo(socket, ADR(S_BUF.BUFFER[s_cur_pos]), s_cur_size, 0, ADR(sockaddr), SIZEOF(sockaddr), ADR(pResult));
	ELSE
		bytes_sent := SysSockSend(socket, ADR(S_BUF.BUFFER[s_cur_pos]), s_cur_size, 0, ADR(pResult));
	END_IF;

	CASE bytes_sent OF
	-2147483648..-1:	; (* ERROR: Noch nicht bereit um Daten aufzunehmen -> nächsten Zyklus wieder probieren *)
	 0: IF NOT udp_mode THEN (* TCP-Mode: socket wurde von remote geschlossen *)
			c_status := 253;
			c_ready := FALSE;
		END_IF;
	ELSE
		s_done := TRUE;
		s_cur_size := DINT_TO_INT(bytes_sent); (* Anzahl der wirklich versendeten Bytes übernehmen *)
		(* ---------------------- Debug-Message ----------------------------*)
		(*IF _debug_enable THEN
			LOG_CL.NEW_MSG := 'IP_SEN SEND_COUNT ~1 -IP_ID ~6';
			LOG_CL.PRINTF[1] := DINT_TO_STRING(s_cur_size);
			LOG_CL.PRINTF[6] := INT_TO_STRING(debug_ID);
			LOG_MSG();
		END_IF;*)
		(* -----------------------------------------------------------------------------*)
	END_CASE
END_IF;

(* ---------------------------------------------- *)

IF IP_C.R_OBSERVE = FALSE OR s_active THEN
    r_time := tx;
END_IF;

IF c_status = 0 AND tx - c_time > error_time AND c_enable AND NOT c_ready AND c_mode < 2 THEN (* Connect Timeout *)
	c_status := 255; (* Timeout-Fehler ausgeben *)
END_IF;
IF s_status = 0 AND tx - s_time > error_time AND s_active THEN (* Send Timeout *)
	s_status := 255; (* Timeout-Fehler ausgeben *)
END_IF;
IF r_status = 0 AND tx - r_time > error_time AND c_ready AND IP_C.R_OBSERVE THEN (* Receive Timeout *)
	r_status := 255; (* Timeout-Fehler ausgeben *)
END_IF;

IP_C.ERROR := OSCAT_BASIC.DWORD_OF_BYTE(c_status,s_status,r_status,0);

(* ---------------------- Debug-Message ----------------------------*)
(*IF  _debug_enable THEN
	IF (IP_C.ERROR <> debug_lasterror) THEN
		LOG_CL.NEW_MSG := 'IP_ERROR ~1 -IP_ID ~6';
		LOG_CL.PRINTF[1] := DWORD_TO_STRING(IP_C.ERROR);
		LOG_CL.PRINTF[6] := INT_TO_STRING(debug_ID);
		LOG_MSG();

		debug_lasterror := IP_C.ERROR;
		debug_last_id := debug_ID;
	END_IF;
END_IF;*)
(* -----------------------------------------------------------------------------*)

(* revision history
ks	18. oct. 2008	rev 1.0
	original version
ks	05. jan. 2009	rev 1.1
	zusätzlichen Parameter "Port" hinzugefügt, und Code bei Verbindungsaufbau angepasst
ks	28. feb. 2009	rev 1.2
	connect code angepasst und verkürzung der zyklen bei Send
ks	20. oct. 2009	rev 1.3
	network_buffer basis 0
ks	06. dec. 2009	rev 1.4
	receive_count MAILBOX[1]
ks	10. nov. 2010	rev 1.5
	send_pause MAILBOX[2] and receive_pause MAILBOX[3] 
ks	07. feb. 2011	rev 1.6
	Fehlercode 253 bei Remote-Verbindungsabbruch
ks	30. may. 2011	rev 1.7
	Fehler bei Empfangsüberwachung
ks	26. july. 2011	rev 1.8
	Error-Reset, diverse optimierungen 
ks	26. feb. 2012	rev 1.9
	Code-Optimierung für höhere kompatibilität

*)

END_FUNCTION_BLOCK

// Common/Function Blocks/IP_CONTROL_135_1
FUNCTION_BLOCK IP_CONTROL_135_1

VAR_IN_OUT
	IP_C : IP_C; (* IP_Control Verwaltungsstruktur *)
	S_BUF : NETWORK_BUFFER; (* Externer Sendbuffer *)
	R_BUF : NETWORK_BUFFER; (* Externer Receivebuffer *)
END_VAR
VAR_INPUT
	IP : DWORD; (* IP Adresse *)
	PORT : WORD; (* Port Nummer *)
	TIME_OUT : TIME; (* Ueberwachungszeit Connect / Send / Receive *)
END_VAR
VAR
	c_time : UDINT; (* CONNECT-Time (Zeit bei nicht vorhandener Verbindung) *)
	s_time : UDINT; (* SEND-Time    (Zeit seit letzten Datensenden) *)
	r_time : UDINT; (* RECEIVE-Time (Zeit seit letztem Datenempfang) *)

	c_enable : BOOL; (* Connect: freigabe *)
	c_ip : DWORD; (* Connect: aktuelle IP-Adresse *)
	c_port : WORD; (* Connect: aktuelle Port-Nummer *)
	c_mode : BYTE; (* Connect: aktueller Mode UDP/TCP...... *)
	c_status : BYTE; (* Connect: Status (Errorcode) *)
	c_ready : BOOL; (* Connect: Verbindung aufgebaut *)
	c_ready_old : BOOL; (* Connect: letzter Zustand von c_ready für Flankenauswertung *)
	c_select : BOOL; (* non blocking mode - abfrage über select durchführen *)
	c_fdWrite : SOCKET_FD_SET;
	c_Timeout : SOCKET_TIMEVAL;

	s_total : INT; (* Send: Gesamtanzahl Bytes zum senden *)
	s_cur_pos : INT; (* Send: aktuelle Sendeposition *)
	s_cur_size : INT; (* Send: aktuelle Sendegroesse *)
	s_max_size : INT; (* Send: maximale Telegrammlänge fuer Senden *)
	s_start : BOOL; (* Send: Sende modus aktivieren *)
	s_active : BOOL; (* Send: Daten senden ist aktiv *)
	s_req : BOOL; (* Send: Start Daten senden *)
	s_done : BOOL; (* Send: ohne Fehler beendet *)
	s_status : BYTE; (* Send: Status (Errorcodes) *)

	r_status : BYTE; (* Receive: Status (Errorcodes) *)
	r_count : INT; (* Receive: Anzahl empfangener Bytes *)
	r_offset : INT; (* Receive: aktuelle Position in externen Receivebuffer *)
	r_max_size : INT; (* Receive: groesse des externen Empfangbuffers*)

	new_connection : BOOL; (* Neue Verbindungsparameter vorhanden *)
	tx : DWORD; (* letzter zeitwert *)
	error_time : DWORD; (* aktueller Timeout-Wert *)

	state: BYTE; (* schrittmerker für connect *)
	server_socket : RTS_IEC_HANDLE:= RTS_INVALID_HANDLE; 
	socket : RTS_IEC_HANDLE:= RTS_INVALID_HANDLE;
	sockaddr : SOCKADDRESS;
	sockaddr_size : DWORD;
	plc_841 : BOOL;
	plc_881 : BOOL;
	dint_true : DINT := 1;
	bytes_received : DINT;
	bytes_sent : DINT;
	udp_mode : BOOL;
	pResult : UDINT; //Needed for V3 Lib
	(*LOG_MSG : LOG_MSG;
	_debug_enable : BOOL := TRUE;
	debug_index : INT;
	debug_ID : INT;
	debug_lasterror : DWORD;
	debug_last_id : INT := 255;
	state_last: BYTE;*)

END_VAR

VAR CONSTANT
	STOP : BYTE := 0;
	TS_INIT: BYTE := 1;
	TS_OPEN : BYTE:= 2;

	UDP_INIT : BYTE:= 31;

	TC_INIT : BYTE:= 51;
	TC_CONNECT : BYTE:= 52;

	C_WAIT : BYTE:= 250;
	C_CLOSE : BYTE:= 251;

END_VAR

(*

version 1.9		26. Feb. 2012
programmer 		ks
tested by			ks

IP_CONTROL ist ein Wrapper-Baustein um eine Hersteller neutrale Schnittstelle zum Ethernet zu schaffen
*)

(* ---------------------- Debug-Message ----------------------------*)
(*IF _debug_enable THEN
	IF IP_C.FIFO.ID > BYTE#0 THEN
		debug_index := IP_C.FIFO.NR;
		debug_ID := BYTE_TO_INT(IP_C.FIFO.X[debug_index]);
	END_IF;
END_IF;*)
(* -----------------------------------------------------------------------------*)

(* read system time *)
tx := OSCAT_BASIC.T_PLC_MS();

IF IP_C.C_PORT = 0 THEN
	IP_C.C_PORT := PORT; (* uebergebenen PORT durch parametrierten PORT ersetzen *)
END_IF;
IF IP_C.C_IP = 0 AND IP_C.C_MODE < 4 THEN
	IP_C.C_IP := IP; (* uebergebene IP durch paramtrierte IP ersetzen *)
END_IF;

new_connection := c_ip <> IP_C.C_IP OR c_mode <> IP_C.C_MODE OR c_port <> IP_C.C_PORT; (* neue Verbindungs erwünscht ? *)
c_enable := IP_C.C_ENABLE AND NOT new_connection;

IF IP_C.C_ENABLE AND IP_C.ERROR = 0 AND state = STOP THEN (* Freigabe,kein Fehler,kein Socket offen *)
	c_ip   := IP_C.C_IP;
	c_mode := IP_C.C_MODE;
	c_port := IP_C.C_PORT;
	plc_841 := SYSLIBSOCKETS_OPTION.1; (* Bit 1 = WAGO 750-841 *)
	plc_881 := SYSLIBSOCKETS_OPTION.2; (* Bit 1 = WAGO 750-881 *)
	udp_mode := C_MODE.0; (* Mode 1,3,5 = udp *)

	error_time := TIME_TO_DWORD(MAX(T#200ms,TIME_OUT));
	IP_C.TIME_RESET := TRUE; (* Alle Timer ruecksetzen *)

	r_max_size := SIZEOF(R_BUF.BUFFER);
	s_max_size := SIZEOF(S_BUF.BUFFER);

	IF C_MODE.0 THEN (* Mode: 1,3,5 = UDP CLIENT/SERVER *)
		state := UDP_INIT;
	ELSIF C_MODE = 0 THEN (* Mode: 0 = TCP CLIENT *)
		state := TC_INIT;
	ELSE
		state := TS_INIT; (* Mode: 2,4 = TCP SERVER *)
	END_IF;

	(* ---------------------- Debug-Message ----------------------------*)
	(*IF _debug_enable THEN
		LOG_CL.NEW_MSG := 'IP_CON: MODE ~1 / IP ~2 / PORT ~3 /ID ~6';
		LOG_CL.PRINTF[1] := BYTE_TO_STRING(C_MODE);
		LOG_CL.PRINTF[2] := IP4_TO_STRING(c_ip);
		LOG_CL.PRINTF[3] := WORD_TO_STRING(c_port);
		LOG_CL.PRINTF[6] := INT_TO_STRING(debug_ID);
		LOG_MSG();
	END_IF;*)
	(* -----------------------------------------------------------------------------*)

END_IF;

(* ---------------------- Debug-Message ----------------------------*)
(*IF  _debug_enable THEN
	IF state <> state_last THEN
		LOG_CL.NEW_MSG := 'IP_STEP ~1 -IP_ID ~6';
		LOG_CL.PRINTF[1] := BYTE_TO_STRING(state);
		LOG_CL.PRINTF[6] := INT_TO_STRING(debug_ID);
		LOG_MSG();
		state_last := state;
	END_IF;
END_IF;*)
(* -----------------------------------------------------------------------------*)

IF IP_C.TIME_RESET THEN (* Alle Timer ruecksetzen *)
	IP_C.TIME_RESET := FALSE; (* Reset rücksetzen *)
	c_time := tx; (* Connect Timer ruecksetzen *)
	s_time := tx; (* Send Timer ruecksetzen *)
	r_time := tx; (* Receive Timer ruecksetzen *)

	c_status := BYTE#0; (* letzten Connect Fehler rücksetzen *)
	s_status := BYTE#0; (* letzten Send Fehler rücksetzen *)
	r_status := BYTE#0; (* letzten Receive Fehler rücksetzen *)
END_IF;

(* ---------------------------------------------- *)

CASE state OF

UDP_INIT: (* UDP_CLIENT + SERVER *)
	socket := SysSockCreate(SOCKET_AF_INET, SOCKET_DGRAM, SOCKET_IPPROTO_IP, ADR(pResult));
	IF socket < 0 THEN
		c_status := 1; (* SysSockCreate failed *)
		state := C_CLOSE;
	ELSE
		SysSockSetOption(socket, SOCKET_SOL, SOCKET_SO_BROADCAST, ADR(dint_true), SIZEOF(dint_true)); (* allow broadcast *)
		SysSockIoctl(socket, SOCKET_FIONBIO, ADR(dint_true)); (* put socket in non-blocking mode *)
		sockaddr.sin_family := SOCKET_AF_INET;
		sockaddr.sin_port := SysSockHtons(c_port);
		sockaddr.sin_addr.ulAddr := SEL(c_mode = 1, SOCKET_INADDR_ANY, SysSockNtohl(c_ip));

		IF c_mode >= 2 THEN (* SERVER Mode *)
			IF SysSockBind(socket, ADR(sockaddr), SIZEOF(sockaddr)) = 0 THEN
				c_ready := TRUE; (* Connected *)
				state:= C_WAIT;
			ELSE
				c_status := 2; (* SysSockBind failed *)
				state := C_CLOSE;
			END_IF;
		ELSE
			c_ready := TRUE; (* Connected *)
			state:= C_WAIT;
		END_IF;
	END_IF;

(* ---------------------------------------------- *)

TC_INIT: (* TCP-CLIENT (AKTIV) *)
	socket := SysSockCreate(SOCKET_AF_INET, SOCKET_STREAM, SOCKET_IPPROTO_IP, ADR(pResult));
	IF socket < 0 THEN
		c_status := 1;  (* SysSockCreate failed *)
		state := C_CLOSE;
	ELSE
		IF plc_841 OR plc_881 THEN
			SysSockSetOption(socket,6,SOCKET_TCP_NODELAY, ADR(dint_true), SIZEOF(dint_true)); (* Set Push-Bit *)
		END_IF;
		SysSockIoctl(socket, SOCKET_FIONBIO, ADR(dint_true)); (* NonBlocking mode *)
		sockaddr.sin_family := SOCKET_AF_INET;
		sockaddr.sin_port := SysSockNtohs(c_port);
		sockaddr.sin_addr.ulAddr := SysSockNtohl(c_ip);
		c_select := FALSE;
		state := TC_CONNECT;
	END_IF;

(* ---------------------------------------------- *)

TC_CONNECT:
	IF NOT c_enable OR c_status = 255 THEN (* keine freigabe oder connect timeout *)
			state:= C_CLOSE;
	ELSE
		IF c_select = FALSE THEN
			IF SysSockConnect(socket,ADR(sockaddr),SIZEOF(sockaddr)) = 0 THEN
				c_ready := TRUE; (* Connected *)
				state:= C_WAIT;
			ELSE
				(* Connect durchgeführt, aber noch nicht verbunden, dann optional mit select-abfrage weitermachen *)
				c_select := SYSLIBSOCKETS_OPTION.0; (* Bit 0 = TCP-Client - use SysSockselect *)
			END_IF;
		ELSE
			c_Timeout.tv_sec := 0;
			c_Timeout.tv_usec := 0;
			c_fdWrite.fd_count := 1;
			c_fdWrite.fd_array[0] := socket;
			IF SysSockSelect(SOCKET_FD_SETSIZE,0,ADR(c_fdWrite),0, ADR(c_Timeout), ADR(pResult)) > 0 THEN
				c_ready := TRUE; (* Connected *)
				state:= C_WAIT;
			END_IF;
		END_IF;
	END_IF;

(* ---------------------------------------------- *)

TS_INIT: (* TCP-SERVER (PASSIV) *)
	server_socket := SysSockCreate(SOCKET_AF_INET, SOCKET_STREAM, SOCKET_IPPROTO_IP, ADR(pResult)); (* Create Socket *)
	IF server_socket = RTS_INVALID_HANDLE THEN
		c_status := 1; (* SysSockCreate failed *)
		state:= C_CLOSE;
	ELSE (* Address bindings *)
		SysSockSetOption( server_socket, SOCKET_SOL, SOCKET_SO_REUSEADDR, ADR(dint_true), SIZEOF(dint_true) );
		sockaddr.sin_family:= SOCKET_AF_INET;
		sockaddr.sin_port := SysSockHtons(c_port);
		sockaddr.sin_addr.ulAddr := SOCKET_INADDR_ANY;
		IF NOT SysSockBind(server_socket, ADR(sockaddr), SIZEOF(sockaddr)) = 0 THEN
			c_status := 2; (* SysSockBind failed *)
			state := C_CLOSE;
		ELSIF NOT SysSockListen(server_socket, 1) = 0 THEN (* erzeugt Warteschlange für eine Verbindung *)
			c_status := 3; (* SysSockListen failed *)
			state:= C_CLOSE;
		ELSE
			SysSockIoctl(server_socket, SOCKET_FIONBIO, ADR(dint_true)); (* NonBlocking mode *)
			state:= TS_OPEN;
		END_IF;
	END_IF;

(* ---------------------------------------------- *)

TS_OPEN: (* Waiting for incomming connection *)
	sockaddr_size := SIZEOF(sockaddr);
	socket := SysSockAccept(server_socket, ADR(sockaddr), ADR(sockaddr_size), ADR(pResult));

	IF socket <> RTS_INVALID_HANDLE THEN (* neuer Verbindungswunsch vorhanden *)
		IF c_mode = BYTE#2 AND sockaddr.sin_addr.ulAddr <> SysSockNtohl(c_ip) THEN (* Mode 2 = TCP + PASSIVE + PORT + IP  auf richtige Partner-IP prüfen *)
			state:= C_CLOSE;
		ELSE
			IF plc_841 OR plc_881 THEN
				SysSockSetOption(socket, 6, SOCKET_TCP_NODELAY, ADR(dint_true), SIZEOF(dint_true)); (* Set Push-Bit *)
			END_IF;
			SysSockIoctl(socket, SOCKET_FIONBIO, ADR(dint_true)); (* NonBlocking mode *)
			c_ready := TRUE; (* Connected *)
			state := C_WAIT;
		END_IF;
	ELSIF NOT c_enable THEN (* keine freigabe mehr ? *)
			state:= C_CLOSE;
	END_IF;

(* ---------------------------------------------- *)

C_WAIT: (* Warten auf Anforderung für Beenden *)
	IF NOT c_enable OR NOT c_ready THEN
		state:= C_CLOSE;
	END_IF

(* ---------------------------------------------- *)

C_CLOSE: (* Close the Sockets *)
	c_ready := FALSE;
	IF socket >= 0 THEN
		IF (NOT plc_841) AND (NOT plc_881) THEN
			SysSockShutdown(socket, 0); (* 870 *)
		END_IF;
		SysSockClose(socket);
		socket := RTS_INVALID_HANDLE;
	END_IF
	IF server_socket >= 0 THEN
		IF (NOT plc_841) AND (NOT plc_881) THEN
			SysSockShutdown(server_socket, 0); (* 870 *)
		END_IF;
		SysSockClose(server_socket);
		server_socket := RTS_INVALID_HANDLE;
	END_IF
	state:= STOP;
END_CASE;

(* ---------------------------------------------- *)

IF c_ready THEN
	IF NOT c_ready_old THEN (* Verbindung aufgebaut - positive Flanke erkannt *)
		IP_C.C_STATE := 254;
		IP_C.TIME_RESET := TRUE; (* Alle Timer ruecksetzen *)
		(* ---------------------- Debug-Message ----------------------------*)
		(*IF _debug_enable THEN
			LOG_CL.NEW_MSG := 'IP_CON: CONNECTED -IP_ID ~6';
			LOG_CL.PRINTF[6] := INT_TO_STRING(debug_ID);
			LOG_MSG();
		END_IF;*)
		(* -----------------------------------------------------------------------------*)
	ELSE
		IP_C.C_STATE := 255; (* Verbindung ist aufgebaut *)
	END_IF;
ELSE
	IF c_ready_old THEN (* Verbindung abgebaut - negative Flanke erkannt *)
		IP_C.C_STATE := 1;
		IP_C.MAILBOX[1] := 0; (* Receive Info rücksetzen *)
		IP_C.MAILBOX[2] := 0; (* Send-Pause rücksetzen *)
		IP_C.MAILBOX[3] := 0; (* Receive-Pause rücksetzen *)
		IF NOT new_connection THEN
			s_active := FALSE; (* Sendeaktivitäten stoppen *)
			s_req := FALSE; (* Sendefreigabe rücksetzen *)
			S_BUF.SIZE := 0; (* Sendelänge löschen *)
			(*IP_C.TIME_RESET := TRUE;*) (* Alle Timer ruecksetzen *)
		END_IF;
		(* ---------------------- Debug-Message ----------------------------*)
		(*IF _debug_enable THEN
			LOG_CL.NEW_MSG := 'IP_CON: DISCONNECTED';
			LOG_MSG();
		END_IF;*)
		(* -----------------------------------------------------------------------------*)
	ELSE
		IP_C.C_STATE := 0; (* Verbindung ist abgebaut *)
	END_IF;
END_IF;

c_ready_old := c_ready;

(* Der Datenempfang wird angehalten solange ein Sendevorgang läuft *)
(* sonst kann es vorkommen das die Antwort-daten schon empfangen werden, *)
(* bevor der Sendevorgang vom programm abgeschlossen wurde *)

IF c_ready AND NOT s_active AND IP_C.MAILBOX[3] = 0 THEN
	IF R_BUF.SIZE >= INT_TO_UINT(r_max_size) THEN
		R_BUF.SIZE := UINT#0;
		r_status := 254; (* Empfangsbuffer wegen Überlauf rückgesetzt *)
	END_IF;

	r_offset := SEL(udp_mode,UINT_TO_INT(R_BUF.SIZE),0);
	r_count := r_max_size - r_offset;

	IF udp_mode THEN
		bytes_received := SysSockRecvFrom(socket, ADR(R_BUF.BUFFER), r_count, 0, ADR(sockaddr), SIZEOF(sockaddr), ADR(pResult));

		IF c_mode = BYTE#3 AND sockaddr.sin_addr.ulAddr <> SysSockNtohl(c_ip) THEN (* Mode 3 = UDP + PASSIVE + PORT + IP  auf richtige Partner-IP prüfen *)
			bytes_received := 0;
			R_BUF.SIZE := UINT#0;
			sockaddr.sin_port := SysSockNtohs(c_port);
			sockaddr.sin_addr.ulAddr := SysSockNtohl(c_ip);
		END_IF;

	ELSE
		bytes_received := SysSockRecv(socket, ADR(R_BUF.BUFFER[r_offset]), r_count, 0, ADR(pResult));
	END_IF;

	(*UDP: IPC returns -1 if no data available or error occured,841 returns -1 if error occured and 0 if no data available*)
	CASE bytes_received OF
	-2147483648..-1: ; (* No data available or error occured *)
	 0: IF NOT udp_mode THEN (* TCP-Mode: socket wurde von remote geschlossen *)
			c_status := 253;
			c_ready := FALSE;
		END_IF;
	ELSE (* daten wurden empfangen *)
  		r_time := tx; (* Receive Timer ruecksetzen *)
		R_BUF.SIZE := INT_TO_UINT(r_offset + DINT_TO_UINT(bytes_received)); (* aktuelle buffersize eintragen *)
		IP_C.MAILBOX[1] := IP_C.MAILBOX[1] + 1; (* Receive Info *)
		IF IP_C.MAILBOX[1] = 0 THEN IP_C.MAILBOX[1] := 1; END_IF;

		(* ---------------------- Debug-Message ----------------------------*)
		(*IF _debug_enable THEN
			LOG_CL.NEW_MSG := 'IP_REC DATA: POS: ~1 : SIZE: ~2 TOTAL ~3 -IP_ID ~6';
			LOG_CL.PRINTF[1] := INT_TO_STRING(r_offset);
			LOG_CL.PRINTF[2] := INT_TO_STRING(r_count);
			LOG_CL.PRINTF[3] := UINT_TO_STRING(R_BUF.SIZE);
			LOG_CL.PRINTF[6] := INT_TO_STRING(debug_ID);
			LOG_MSG();
		END_IF;*)
		(* -----------------------------------------------------------------------------*)

	END_CASE
END_IF;

(* ---------------------------------------------- *)

IF S_BUF.SIZE > 0 THEN
	IF c_ready AND c_enable THEN
		IF NOT s_active AND IP_C.MAILBOX[2] = 0 THEN
			(* Gesamtanzahl an Bytes limitieren und uebergeben *)
			s_total := LIMIT(0,UINT_TO_INT(S_BUF.SIZE),r_max_size);
			s_cur_pos  := 0;
			s_cur_size := 0;
			s_start := TRUE; (* Daten kopieren und senden anstossen *)
			s_active := TRUE; (* Sende-Betrieb aktivieren *)
			(* ---------------------- Debug-Message ----------------------------*)
			(*IF _debug_enable THEN
				LOG_CL.NEW_MSG := 'IP_SEN INIT: TOTAL: ~1 -IP_ID ~6';
				LOG_CL.PRINTF[1] := INT_TO_STRING(S_TOTAL);
				LOG_CL.PRINTF[6] := INT_TO_STRING(debug_ID);
				LOG_MSG();
			END_IF;*)
			(* -----------------------------------------------------------------------------*)
		END_IF;

		IF s_done OR s_start THEN (* Daten senden aktiv *)

			s_start := FALSE;
			s_cur_pos := s_cur_pos + s_cur_size; (* neue Sende-Datenposition bestimmen *)
			IF s_total > s_cur_pos THEN (* weitere Daten zum senden vorhanden ? *)
				s_cur_size := s_total - s_cur_pos;
				s_cur_size := LIMIT(0, s_cur_size, s_max_size); (* Telegrammlänge begrenzen *)
				(* ---------------------- Debug-Message ----------------------------*)
				(*IF _debug_enable THEN
					LOG_CL.NEW_MSG := 'IP_SEN DATA: POS: ~1 : SIZE: ~2 TOTAL ~3 -IP_ID ~6';
					LOG_CL.PRINTF[1] := INT_TO_STRING(S_CUR_POS);
					LOG_CL.PRINTF[2] := INT_TO_STRING(S_CUR_SIZE);
					LOG_CL.PRINTF[3] := INT_TO_STRING(S_TOTAL);
					LOG_CL.PRINTF[6] := INT_TO_STRING(debug_ID);
					LOG_MSG();
				END_IF;*)
				(* -----------------------------------------------------------------------------*)
				s_time := tx; (* Send Timer ruecksetzen *)
				r_time := tx; (* Receive Timer ruecksetzen *)
				s_req := TRUE;

			ELSE
				(* keine weitere Sendedaten vorhanden -> Senden beenden *)
				s_req := FALSE;
				s_active := FALSE;
				S_BUF.SIZE := 0;
				(* ---------------------- Debug-Message ----------------------------*)
				(*IF _debug_enable THEN
					LOG_CL.NEW_MSG := 'IP_SEN FINISH -IP_ID ~6';
					LOG_CL.PRINTF[6] := INT_TO_STRING(debug_ID);
					LOG_MSG();
				END_IF;*)
				(* -----------------------------------------------------------------------------*)
			END_IF;
		END_IF;
	END_IF;
END_IF;

IF s_req THEN
	s_done := FALSE;
	IF udp_mode THEN
		bytes_sent := SysSockSendTo(socket, ADR(S_BUF.BUFFER[s_cur_pos]), s_cur_size, 0, ADR(sockaddr), SIZEOF(sockaddr), ADR(pResult));
	ELSE
		bytes_sent := SysSockSend(socket, ADR(S_BUF.BUFFER[s_cur_pos]), s_cur_size, 0, ADR(pResult));
	END_IF;

	CASE bytes_sent OF
	-2147483648..-1:	; (* ERROR: Noch nicht bereit um Daten aufzunehmen -> nächsten Zyklus wieder probieren *)
	 0: IF NOT udp_mode THEN (* TCP-Mode: socket wurde von remote geschlossen *)
			c_status := 253;
			c_ready := FALSE;
		END_IF;
	ELSE
		s_done := TRUE;
		s_cur_size := DINT_TO_INT(bytes_sent); (* Anzahl der wirklich versendeten Bytes übernehmen *)
		(* ---------------------- Debug-Message ----------------------------*)
		(*IF _debug_enable THEN
			LOG_CL.NEW_MSG := 'IP_SEN SEND_COUNT ~1 -IP_ID ~6';
			LOG_CL.PRINTF[1] := DINT_TO_STRING(s_cur_size);
			LOG_CL.PRINTF[6] := INT_TO_STRING(debug_ID);
			LOG_MSG();
		END_IF;*)
		(* -----------------------------------------------------------------------------*)
	END_CASE
END_IF;

(* ---------------------------------------------- *)

IF IP_C.R_OBSERVE = FALSE OR s_active THEN
    r_time := tx;
END_IF;

IF c_status = 0 AND tx - c_time > error_time AND c_enable AND NOT c_ready AND c_mode < 2 THEN (* Connect Timeout *)
	c_status := 255; (* Timeout-Fehler ausgeben *)
END_IF;
IF s_status = 0 AND tx - s_time > error_time AND s_active THEN (* Send Timeout *)
	s_status := 255; (* Timeout-Fehler ausgeben *)
END_IF;
IF r_status = 0 AND tx - r_time > error_time AND c_ready AND IP_C.R_OBSERVE THEN (* Receive Timeout *)
	r_status := 255; (* Timeout-Fehler ausgeben *)
END_IF;

IP_C.ERROR := OSCAT_BASIC.DWORD_OF_BYTE(c_status,s_status,r_status,0);

(* ---------------------- Debug-Message ----------------------------*)
(*IF  _debug_enable THEN
	IF (IP_C.ERROR <> debug_lasterror) THEN
		LOG_CL.NEW_MSG := 'IP_ERROR ~1 -IP_ID ~6';
		LOG_CL.PRINTF[1] := DWORD_TO_STRING(IP_C.ERROR);
		LOG_CL.PRINTF[6] := INT_TO_STRING(debug_ID);
		LOG_MSG();

		debug_lasterror := IP_C.ERROR;
		debug_last_id := debug_ID;
	END_IF;
END_IF;*)
(* -----------------------------------------------------------------------------*)

(* revision history
ks	18. oct. 2008	rev 1.0
	original version
ks	05. jan. 2009	rev 1.1
	zusätzlichen Parameter "Port" hinzugefügt, und Code bei Verbindungsaufbau angepasst
ks	28. feb. 2009	rev 1.2
	connect code angepasst und verkürzung der zyklen bei Send
ks	20. oct. 2009	rev 1.3
	network_buffer basis 0
ks	06. dec. 2009	rev 1.4
	receive_count MAILBOX[1]
ks	10. nov. 2010	rev 1.5
	send_pause MAILBOX[2] and receive_pause MAILBOX[3] 
ks	07. feb. 2011	rev 1.6
	Fehlercode 253 bei Remote-Verbindungsabbruch
ks	30. may. 2011	rev 1.7
	Fehler bei Empfangsüberwachung
ks	26. july. 2011	rev 1.8
	Error-Reset, diverse optimierungen 
ks	26. feb. 2012	rev 1.9
	Code-Optimierung für höhere kompatibilität

*)

END_FUNCTION_BLOCK

// Common/Function Blocks/IP_CONTROL_old
FUNCTION_BLOCK IP_CONTROL_old
VAR_IN_OUT
	IP_C : IP_C; (* IP_Control Verwaltungsstruktur *)
	S_BUF : NETWORK_BUFFER; (* Externer Sendbuffer *)
	R_BUF : NETWORK_BUFFER; (* Externer Receivebuffer *)
END_VAR
VAR_INPUT
	IP : DWORD; (* IP Adresse *)
	PORT : WORD; (* Port Nummer *)
	TIME_OUT : TIME; (* Ueberwachungszeit Connect / Send / Receive *)
END_VAR
VAR
	c_time : UDINT; (* CONNECT-Time (Zeit bei nicht vorhandener Verbindung) *)
	s_time : UDINT; (* SEND-Time    (Zeit seit letzten Datensenden) *)
	r_time : UDINT; (* RECEIVE-Time (Zeit seit letztem Datenempfang) *)

	c_enable : BOOL; (* Connect: freigabe *)
	c_ip : DWORD; (* Connect: aktuelle IP-Adresse *)
	c_port : WORD; (* Connect: aktuelle Port-Nummer *)
	c_mode : BYTE; (* Connect: aktueller Mode UDP/TCP...... *)
	c_status : BYTE; (* Connect: Status (Errorcode) *)
	c_ready : BOOL; (* Connect: Verbindung aufgebaut *)
	c_ready_old : BOOL; (* Connect: letzter Zustand von c_ready für Flankenauswertung *)
	c_select : BOOL; (* non blocking mode - abfrage über select durchführen *)
	c_fdWrite : SOCKET_FD_SET;
	c_Timeout : SOCKET_TIMEVAL;

	s_total : INT; (* Send: Gesamtanzahl Bytes zum senden *)
	s_cur_pos : INT; (* Send: aktuelle Sendeposition *)
	s_cur_size : INT; (* Send: aktuelle Sendegroesse *)
	s_max_size : INT; (* Send: maximale Telegrammlänge fuer Senden *)
	s_start : BOOL; (* Send: Sende modus aktivieren *)
	s_active : BOOL; (* Send: Daten senden ist aktiv *)
	s_req : BOOL; (* Send: Start Daten senden *)
	s_done : BOOL; (* Send: ohne Fehler beendet *)
	s_status : BYTE; (* Send: Status (Errorcodes) *)

	r_status : BYTE; (* Receive: Status (Errorcodes) *)
	r_count : INT; (* Receive: Anzahl empfangener Bytes *)
	r_offset : INT; (* Receive: aktuelle Position in externen Receivebuffer *)
	r_max_size : INT; (* Receive: groesse des externen Empfangbuffers*)

	new_connection : BOOL; (* Neue Verbindungsparameter vorhanden *)
	tx : DWORD; (* letzter zeitwert *)
	error_time : DWORD; (* aktueller Timeout-Wert *)

	state: BYTE; (* schrittmerker für connect *)
	server_socket : RTS_IEC_HANDLE:= RTS_INVALID_HANDLE;                // Handle Pointing to our Socket
	socket : RTS_IEC_HANDLE:= RTS_INVALID_HANDLE;
	//server_socket : DINT:= RTS_INVALID_HANDLE;
	//socket : DINT:= RTS_INVALID_HANDLE;
	sockaddr : SOCKADDRESS;
	sockaddr_size : DWORD;
	plc_841 : BOOL;
	plc_881 : BOOL;
	dint_true : DINT := 1;
	bytes_received : DINT;
	bytes_sent : DINT;
	udp_mode : BOOL;

	pResult : UDINT; //Needed for V3 Lib
	FunctionResult 	: UDINT ;   
  	tAddress                	: INADDR;                           // Strucutre to define our internet address
	TESTtAddress               	: INADDR;   
	(*LOG_MSG : LOG_MSG;
	_debug_enable : BOOL := TRUE;
	debug_index : INT;
	debug_ID : INT;
	debug_lasterror : DWORD;
	debug_last_id : INT := 255;
	state_last: BYTE;*)


END_VAR

VAR CONSTANT
	STOP : BYTE := 0;
	TS_INIT: BYTE := 1;
	TS_OPEN : BYTE:= 2;

	UDP_INIT : BYTE:= 31;

	TC_INIT : BYTE:= 51;
	TC_CONNECT : BYTE:= 52;

	C_WAIT : BYTE:= 250;
	C_CLOSE : BYTE:= 251;

END_VAR

(*

version 1.9		26. Feb. 2012
programmer 		ks
tested by			ks

IP_CONTROL ist ein Wrapper-Baustein um eine Hersteller neutrale Schnittstelle zum Ethernet zu schaffen
*)

(* ---------------------- Debug-Message ----------------------------*)
(*IF _debug_enable THEN
	IF IP_C.FIFO.ID > BYTE#0 THEN (* nur wenn Teilnehmer ID's vorhanden sind *)
		debug_index := IP_C.FIFO.NR;
		debug_ID := BYTE_TO_INT(IP_C.FIFO.X[debug_index]);
	END_IF;
END_IF;*)
(* -----------------------------------------------------------------------------*)

(* read system time *)
tx := OSCAT_BASIC.T_PLC_MS();

IF IP_C.C_PORT = 0 THEN
	IP_C.C_PORT := PORT; (* uebergebenen PORT durch parametrierten PORT ersetzen *)
END_IF;
IF IP_C.C_IP = 0 AND IP_C.C_MODE < 4 THEN
	IP_C.C_IP := IP; (* uebergebene IP durch paramtrierte IP ersetzen *)
END_IF;

new_connection := c_ip <> IP_C.C_IP OR c_mode <> IP_C.C_MODE OR c_port <> IP_C.C_PORT; (* neue Verbindungs erwünscht ? *)
c_enable := IP_C.C_ENABLE AND NOT new_connection;

IF IP_C.C_ENABLE AND IP_C.ERROR = 0 AND state = STOP THEN (* Freigabe,kein Fehler,kein Socket offen *)
	c_ip   := IP_C.C_IP;
	c_mode := IP_C.C_MODE;
	c_port := IP_C.C_PORT;
	plc_841 := ADR(%MW0)=16#30000000; (*750-841*)
	plc_881 := ADR(%MW0)=16#20000000; (*750-881*)
	udp_mode := C_MODE.0; (* Mode 1,3,5 = udp *)

	error_time := TIME_TO_DWORD(MAX(T#200ms,TIME_OUT));
	IP_C.TIME_RESET := TRUE; (* Alle Timer ruecksetzen *)

	r_max_size := UINT_TO_INT(SIZEOF(R_BUF.BUFFER));
	s_max_size := UINT_TO_INT(SIZEOF(S_BUF.BUFFER));

	IF C_MODE.0 THEN (* Mode: 1,3,5 = UDP CLIENT/SERVER *)
		state := UDP_INIT;
	ELSIF C_MODE = 0 THEN (* Mode: 0 = TCP CLIENT *)
		state := TC_INIT;
	ELSE
		state := TS_INIT; (* Mode: 2,4 = TCP SERVER *)
	END_IF;

	(* ---------------------- Debug-Message ----------------------------*)
	(*IF _debug_enable THEN
		LOG_CL.NEW_MSG := 'IP_CON: MODE ~1 / IP ~2 / PORT ~3 /ID ~6';
		LOG_CL.PRINTF[1] := BYTE_TO_STRING(C_MODE);
		LOG_CL.PRINTF[2] := IP4_TO_STRING(c_ip);
		LOG_CL.PRINTF[3] := WORD_TO_STRING(c_port);
		LOG_CL.PRINTF[6] := INT_TO_STRING(debug_ID);
		LOG_MSG();
	END_IF;*)
	(* -----------------------------------------------------------------------------*)

END_IF;

(* ---------------------- Debug-Message ----------------------------*)
(*IF  _debug_enable THEN
	IF state <> state_last THEN
		LOG_CL.NEW_MSG := 'IP_STEP ~1 -IP_ID ~6';
		LOG_CL.PRINTF[1] := BYTE_TO_STRING(state);
		LOG_CL.PRINTF[6] := INT_TO_STRING(debug_ID);
		LOG_MSG();
		state_last := state;
	END_IF;
END_IF;*)
(* -----------------------------------------------------------------------------*)

IF IP_C.TIME_RESET THEN (* Alle Timer ruecksetzen *)
	IP_C.TIME_RESET := FALSE; (* Reset rücksetzen *)
	c_time := tx; (* Connect Timer ruecksetzen *)
	s_time := tx; (* Send Timer ruecksetzen *)
	r_time := tx; (* Receive Timer ruecksetzen *)

	c_status := BYTE#0; (* letzten Connect Fehler rücksetzen *)
	s_status := BYTE#0; (* letzten Send Fehler rücksetzen *)
	r_status := BYTE#0; (* letzten Receive Fehler rücksetzen *)
END_IF;

(* ---------------------------------------------- *)

CASE state OF

